// TIA Portal project "Pierwszy_Projekt_16022023" (V16)

(* hardware
DEVICE "S71500/ET200MP station_1"  S7-1500 station
   slot 0: "Rail_0"  Rack  6ES7 590-1***0-0AA0
   slot 1: "PLC_1"  CPU 1518F-4 PN/DP  6ES7 518-4FP00-3AB0  V2.8
      slot 3: "CPU display_1"  6ES7591-1BA00-0AA0
      slot 32768: "PROFINET interface_1"  X1
         slot 32769: "Port_1"  X1 P1
         slot 32770: "Port_2"  X1 P2
      slot 33024: "PROFINET interface_2"  X2
         slot 33025: "Port_1"  X2 P1
      slot 33280: "PROFINET interface GBIT_3"  X3
         slot 33281: "Port_1"  X3 P1
      slot 33536: "DP interface_1"  X4
      slot 34817: "Virtual CP interface port_1"  Virtual CP interface port  Virtual CP interface port
*)

// ===== PLC "PLC_1"  CPU 1518F-4 PN/DP =====

VAR_GLOBAL   // PLC tag table "Default tag table"
   "System_Byte" AT %MB1 : Byte;
   "FirstScan" AT %M1.0 : Bool;
   "DiagStatusUpdate" AT %M1.1 : Bool;
   "AlwaysTRUE" AT %M1.2 : Bool;
   "AlwaysFALSE" AT %M1.3 : Bool;
   "Clock_Byte" AT %MB0 : Byte;
   "Clock_10Hz" AT %M0.0 : Bool;
   "Clock_5Hz" AT %M0.1 : Bool;
   "Clock_2.5Hz" AT %M0.2 : Bool;
   "Clock_2Hz" AT %M0.3 : Bool;
   "Clock_1.25Hz" AT %M0.4 : Bool;
   "Clock_1Hz" AT %M0.5 : Bool;
   "Clock_0.625Hz" AT %M0.6 : Bool;
   "Clock_0.5Hz" AT %M0.7 : Bool;
   "11-PLC01-MANUAL" AT %Q1.6 : Bool;
   "11-PLC01-AUTOMAT" AT %Q1.7 : Bool;
   "11-PLC01-DISPLAY01" AT %QD58 : Real;
   "Tag_1" AT %QD40 : Real;
   "Tag_2" AT %Q2.5 : Bool;
   "Tag_3" AT %QD48 : Real;
   "Tag_4" AT %M2.0 : Bool;
   "Tag_5" AT %I4.4 : Bool;
   "Tag_6" AT %M3.0 : Bool;
   "Tag_7" AT %M3.1 : Bool;
   "Tag_8" AT %M3.2 : Bool;
END_VAR

VAR_GLOBAL   // PLC tag table "Tag table from XML_1"
   "11-PLC01-CNR01-SQ01" AT %I0.0 : Bool;
   "11-PLC01-CNR01-SQ02" AT %I0.1 : Bool;
   "11-PLC01-CNR01-ENC-A" AT %I0.2 : Bool;
   "11-PLC01-CNR01-ENC-B" AT %I0.3 : Bool;
   "11-PLC01-CNR02-SQ01" AT %I0.4 : Bool;
   "11-PLC01-CNR02-SQ02" AT %I0.5 : Bool;
   "11-PLC01-CNR02-ENC-A" AT %I0.6 : Bool;
   "11-PLC01-CNR02-ENC-B" AT %I0.7 : Bool;
   "11-PLC01-CNR03-SQ01" AT %I1.0 : Bool;
   "11-PLC01-CNR03-SQ02" AT %I1.1 : Bool;
   "11-PLC01-CNR03-ENC-A" AT %I1.2 : Bool;
   "11-PLC01-CNR03-ENC-B" AT %I1.3 : Bool;
   "11-PLC01-B01(START)" AT %I3.5 : Bool;
   "11-PLC01-B02(STOP)" AT %I3.6 : Bool;
   "11-PLC01-B03(RESET)" AT %I3.7 : Bool;
   "11-PLC01-B04(MANUAL)" AT %I4.0 : Bool;
   "11-PLC01-B05(AUTOMAT)" AT %I4.1 : Bool;
   "FACTORY I/O (Running)" AT %I4.2 : Bool;
   "FACTORY I/O (Paused)" AT %I4.3 : Bool;
   "FACTORY I/O (Reset)" AT %Q1.5 : Bool;
   "11-PLC01-PX01(START)" AT %Q0.0 : Bool;
   "11-PLC01-PX02(STOP)" AT %Q0.1 : Bool;
   "11-PLC01-PX03(RESET)" AT %Q0.2 : Bool;
   "11-PLC01-CNR01-EM01" AT %Q0.3 : Bool;
   "11-PLC01-CNR03-RE01" AT %Q0.4 : Bool;
   "FACTORY I/O (Run)" AT %Q1.3 : Bool;
   "FACTORY I/O (Pause)" AT %Q1.4 : Bool;
   "FACTORY I/O (Time Scale)" AT %ID34 : Real;
   "11-PLC01-CNR01" AT %QD30 : Real;
   "11-PLC01-CNR02" AT %QD34 : Real;
   "11-PLC01-CNR03" AT %QD38 : Real;
   "FACTORY I/O (Camera Position)" AT %QD54 : DInt;
   "11-PLC01-TT01-SQ01" AT %I1.4 : Bool;
   "11-PLC01-TT01-SQ02" AT %I1.5 : Bool;
   "11-PLC01-TT01-SQ03" AT %I1.6 : Bool;
   "11-PLC01-TT01-SQ04" AT %I1.7 : Bool;
   "11-PLC01-TT01-SQ05" AT %I2.0 : Bool;
   "11-PLC01-CNR04-SQ01" AT %I2.1 : Bool;
   "11-PLC01-CNR04-SQ02" AT %I2.2 : Bool;
   "11-PLC01-CNR04-ENC-A" AT %I2.3 : Bool;
   "11-PLC01-CNR04-ENC-B" AT %I2.4 : Bool;
   "11-PLC01-CNR05-SQ01" AT %I2.5 : Bool;
   "11-PLC01-CNR05-SQ02" AT %I2.6 : Bool;
   "11-PLC01-CNR05-ENC-A" AT %I2.7 : Bool;
   "11-PLC01-CNR05-ENC-B" AT %I3.0 : Bool;
   "11-PLC01-CNR06-SQ01" AT %I3.1 : Bool;
   "11-PLC01-CNR06-SQ02" AT %I3.2 : Bool;
   "11-PLC01-CNR06-ENC-A" AT %I3.3 : Bool;
   "11-PLC01-CNR06-ENC-B" AT %I3.4 : Bool;
   "11-PLC01-CNR04-RE01" AT %Q0.5 : Bool;
   "11-PLC01-CNR05-RE01" AT %Q0.6 : Bool;
   "11-PLC01-CNR06-RE01" AT %Q0.7 : Bool;
   "11-PLC01-TT01-LEFT" AT %Q2.0 : Bool;
   "11-PLC01-TT01-RIGHT" AT %Q2.1 : Bool;
   "11-PLC01-TT01-FORWARD" AT %Q2.2 : Bool;
   "11-PLC01-TT01-BACKWARD" AT %Q2.3 : Bool;
   "11-PLC01-CNR03-FLC01" AT %ID30 : Real;
   "11-PLC01-CNR04" AT %QD42 : Real;
   "11-PLC01-CNR05" AT %QD46 : Real;
   "11-PLC01-CNR06" AT %QD50 : Real;
END_VAR

DATA_BLOCK "Main_Safety_RTG1_DB"   // DB1, F_DB
{ S7_Optimized_Access := 'TRUE' }
NAME : FUSI
VERSION : 0.1
// stored: InstanceOfName Main_Safety_RTG1
"Main_Safety_RTG1"
BEGIN
END_DATA_BLOCK

DATA_BLOCK "IDB_11_CNR01"   // DB4
{ S7_Optimized_Access := 'TRUE' }
VERSION : 0.1
// stored: InstanceOfName FB_Conveyor
"FB_Conveyor"
BEGIN
END_DATA_BLOCK

DATA_BLOCK "IDB_11_CNR02"   // DB5
{ S7_Optimized_Access := 'TRUE' }
VERSION : 0.1
// stored: InstanceOfName FB_Conveyor
"FB_Conveyor"
BEGIN
END_DATA_BLOCK

DATA_BLOCK "DB_Manual"   // DB6
{ S7_Optimized_Access := 'TRUE' }
VERSION : 0.1
   VAR
      "11-CNR01-CONV" : Struct
         SelectManualMode : Bool := TRUE;
         StartStop : Bool := TRUE;
         SetSpeed : Int := 33;
      END_STRUCT;
      "11-CNR02-CONV" : Struct
         SelectManualMode : Bool := TRUE;
         StartStop : Bool := TRUE;
         SetSpeed : Int := 66;
      END_STRUCT;
      "11-CNR03-CONV" : Struct
         SelectManualMode : Bool := TRUE;
         StartStop : Bool := TRUE;
         SetSpeed : Int := 99;
      END_STRUCT;
   END_VAR
BEGIN
END_DATA_BLOCK

DATA_BLOCK "IDB_11_CNR03"   // DB7
{ S7_Optimized_Access := 'TRUE' }
VERSION : 0.1
// stored: InstanceOfName FB_Conveyor
"FB_Conveyor"
BEGIN
END_DATA_BLOCK

DATA_BLOCK "IDB_11_CNR01_VFD"   // DB8
{ S7_Optimized_Access := 'TRUE' }
VERSION : 0.1
// stored: InstanceOfName FB_Inverter
"FB_Inverter"
BEGIN
END_DATA_BLOCK

DATA_BLOCK "DB_Configuration"   // DB9
{ S7_Optimized_Access := 'TRUE' }
VERSION : 0.1
   VAR
      "11-CNR01-VFD_1" : Struct
         InterlockForward : Bool := TRUE;
         InterlockReverse : Bool := FALSE;
      END_STRUCT;
      "11-CNR02-VFD" : Struct
         InterlockForward : Bool := TRUE;
         InterlockReverse : Bool := FALSE;
      END_STRUCT;
      "11-CNR03-VFD" : Struct
         InterlockForward : Bool := TRUE;
         InterlockReverse : Bool := FALSE;
      END_STRUCT;
   END_VAR
BEGIN
END_DATA_BLOCK

DATA_BLOCK "DB_Signals"   // DB10
{ S7_Optimized_Access := 'TRUE' }
VERSION : 0.1
   VAR
      "11-CNR01-VFD" : Struct
         RunForward : Bool;
         RunReverse : Bool;
         ConveyorSpeedSetpoint : Real := 0.0;
      END_STRUCT;
      "11-CNR02-VFD" : Struct
         RunForward : Bool;
         RunReverse : Bool;
         ConveyorSpeedSetpoint : Real := 0.0;
      END_STRUCT;
      "11-CNR03-VFD" : Struct
         RunForward : Bool;
         RunReverse : Bool;
         ConveyorSpeedSetpoint : Real := 0.0;
      END_STRUCT;
   END_VAR
BEGIN
END_DATA_BLOCK

DATA_BLOCK "IDB_11_CNR02_VFD"   // DB11
{ S7_Optimized_Access := 'TRUE' }
VERSION : 0.1
// stored: InstanceOfName FB_Inverter
"FB_Inverter"
BEGIN
END_DATA_BLOCK

DATA_BLOCK "IDB_11_CNR03_VFD"   // DB12
{ S7_Optimized_Access := 'TRUE' }
VERSION : 0.1
// stored: InstanceOfName FB_Inverter
"FB_Inverter"
BEGIN
END_DATA_BLOCK

DATA_BLOCK "IDB_11_System"   // DB14
{ S7_Optimized_Access := 'TRUE' }
VERSION : 0.1
// stored: InstanceOfName FB_Control
"FB_Control"
BEGIN
END_DATA_BLOCK

DATA_BLOCK "DB_Control"   // DB15
{ S7_Optimized_Access := 'TRUE' }
VERSION : 0.1
   VAR
      StartCommand : Bool := TRUE;
      StopCommand : Bool;
      StartFeedback : Bool;
      StopFeedback : Bool;
      ManualFeedback : Bool;
   END_VAR
BEGIN
END_DATA_BLOCK

DATA_BLOCK "IDB_11_TurnTable"   // DB16
{ S7_Optimized_Access := 'TRUE' }
VERSION : 0.1
// stored: InstanceOfName FB_TurnTable
"FB_TurnTable"
BEGIN
END_DATA_BLOCK

DATA_BLOCK "DB_Chute"   // DB17
{ S7_Optimized_Access := 'TRUE' }
VERSION : 0.1
   VAR
      SmallPackage : Int;
      MediumPackage : Int;
      BigPackage : Int;
   END_VAR
BEGIN
END_DATA_BLOCK

DATA_BLOCK "IDB_Fifo"   // DB18
{ S7_Optimized_Access := 'TRUE' }
VERSION : 0.1
// stored: InstanceOfName FB_Fifo
"FB_Fifo"
BEGIN
END_DATA_BLOCK

DATA_BLOCK "DB_Fifo"   // DB19
{ S7_Optimized_Access := 'TRUE' }
VERSION : 0.1
   VAR
      Array_Destiny : Array[0..10] of Real;
      Array_Return : Int;
      Array_EndOfQueue : Array[0..10] of Real;
      Array_Input : Array[0..5] of Real;
   END_VAR
BEGIN
   Array_Destiny[0] := 0.0;
   Array_Destiny[1] := 0.0;
   Array_Destiny[2] := 0.0;
   Array_Destiny[3] := 0.0;
   Array_Destiny[4] := 0.0;
   Array_Destiny[5] := 0.0;
   Array_Destiny[6] := 0.0;
   Array_Destiny[7] := 0.0;
   Array_Destiny[8] := 0.0;
   Array_Destiny[9] := 0.0;
   Array_Destiny[10] := 0.0;
   Array_EndOfQueue[0] := 0.0;
   Array_EndOfQueue[1] := 0.0;
   Array_EndOfQueue[2] := 0.0;
   Array_EndOfQueue[3] := 0.0;
   Array_EndOfQueue[4] := 0.0;
   Array_EndOfQueue[5] := 0.0;
   Array_EndOfQueue[6] := 0.0;
   Array_EndOfQueue[7] := 0.0;
   Array_EndOfQueue[8] := 0.0;
   Array_EndOfQueue[9] := 0.0;
   Array_EndOfQueue[10] := 0.0;
   Array_Input[0] := 0.0;
   Array_Input[1] := 0.0;
   Array_Input[2] := 0.0;
   Array_Input[3] := 0.0;
   Array_Input[4] := 0.0;
   Array_Input[5] := 0.0;
END_DATA_BLOCK

DATA_BLOCK "IDB_11_CNRO4_AmountOfPackage"   // DB25
{ S7_Optimized_Access := 'TRUE' }
VERSION : 0.1
// stored: InstanceOfName FB_Chute
"FB_Chute"
BEGIN
END_DATA_BLOCK

// folder: System blocks/Program resources

DATA_BLOCK "StartButtonCount_DB"   // DB2
{ S7_Optimized_Access := 'TRUE' }
AUTHOR : Simatic
FAMILY : IEC
NAME : CNTR
VERSION : 1.0
// stored: InstanceOfName IEC_COUNTER
"IEC_COUNTER"
BEGIN
END_DATA_BLOCK

DATA_BLOCK "DelayStart_DB"   // DB3
{ S7_Optimized_Access := 'TRUE' }
AUTHOR : Simatic
FAMILY : IEC
NAME : IEC_TMR
VERSION : 1.0
// stored: InstanceOfName IEC_TIMER
"IEC_TIMER"
BEGIN
END_DATA_BLOCK

DATA_BLOCK "s_TON_Timer"   // DB13
{ S7_Optimized_Access := 'TRUE' }
AUTHOR : Simatic
FAMILY : IEC
NAME : IEC_TMR
VERSION : 1.0
// stored: InstanceOfName IEC_TIMER
"IEC_TIMER"
BEGIN
END_DATA_BLOCK

DATA_BLOCK "IDB_QueueCounter"   // DB21
{ S7_Optimized_Access := 'TRUE' }
AUTHOR : Simatic
FAMILY : IEC
NAME : CNTR
VERSION : 1.0
// stored: InstanceOfName IEC_COUNTER
"IEC_COUNTER"
BEGIN
END_DATA_BLOCK

DATA_BLOCK "IDB_QueueEndCounter"   // DB22
{ S7_Optimized_Access := 'TRUE' }
AUTHOR : Simatic
FAMILY : IEC
NAME : CNTR
VERSION : 1.0
// stored: InstanceOfName IEC_COUNTER
"IEC_COUNTER"
BEGIN
END_DATA_BLOCK

DATA_BLOCK "IEC_Counter_0_DB"   // DB23
{ S7_Optimized_Access := 'TRUE' }
AUTHOR : Simatic
FAMILY : IEC
NAME : CNTR
VERSION : 1.0
// stored: InstanceOfName IEC_COUNTER
"IEC_COUNTER"
BEGIN
END_DATA_BLOCK

DATA_BLOCK "IEC_Counter_0_DB_1"   // DB24
{ S7_Optimized_Access := 'TRUE' }
AUTHOR : Simatic
FAMILY : IEC
NAME : CNTR
VERSION : 1.0
// stored: InstanceOfName IEC_COUNTER
"IEC_COUNTER"
BEGIN
END_DATA_BLOCK

DATA_BLOCK "IEC_Counter_0_DB_2"   // DB26
{ S7_Optimized_Access := 'TRUE' }
AUTHOR : Simatic
FAMILY : IEC
NAME : CNTR
VERSION : 1.0
// stored: InstanceOfName IEC_COUNTER
"IEC_COUNTER"
BEGIN
END_DATA_BLOCK

// folder: (top level)

FUNCTION_BLOCK "Main_Safety_RTG1"   // FB1, F_FBD
{ S7_Optimized_Access := 'TRUE' }
BEGIN
END_FUNCTION_BLOCK

FUNCTION_BLOCK "FB_Conveyor"   // FB2, LAD
{ S7_Optimized_Access := 'TRUE' }
VERSION : 0.1
   VAR_INPUT
      ir_ConveyorSpeed : Real;
      ix_PEC_BOS : Bool;
      ix_PEC_EOS : Bool;
   END_VAR
   VAR_IN_OUT
      iqx_StartStop : Bool;
      iqi_SetSpeed : Int;
      iqx_SelectManualMode : Bool;
      iqx_InverterSpeedSetpoint : Real;
      iqx_InverterRunForward : Bool;
      iqx_InverterRunReverse : Bool;
      iqx_ControlStart : Bool;
      iqx_ControlStop : Bool;
      iqx_ControlManual : Bool;
      igx_ConvFlow : Bool;
   END_VAR
   VAR
      sx_Manual : Bool;
      sx_Automatic : Bool;
   END_VAR
   VAR_TEMP
      tr_SpeedProcent : Real;
   END_VAR
   VAR_TEMP   // added for the SCL form of the ladder/FBD networks
      _w1 : Bool;
      _w2 : Bool;
      _w3 : Bool;
   END_VAR
BEGIN

REGION Network 1: Manual mode
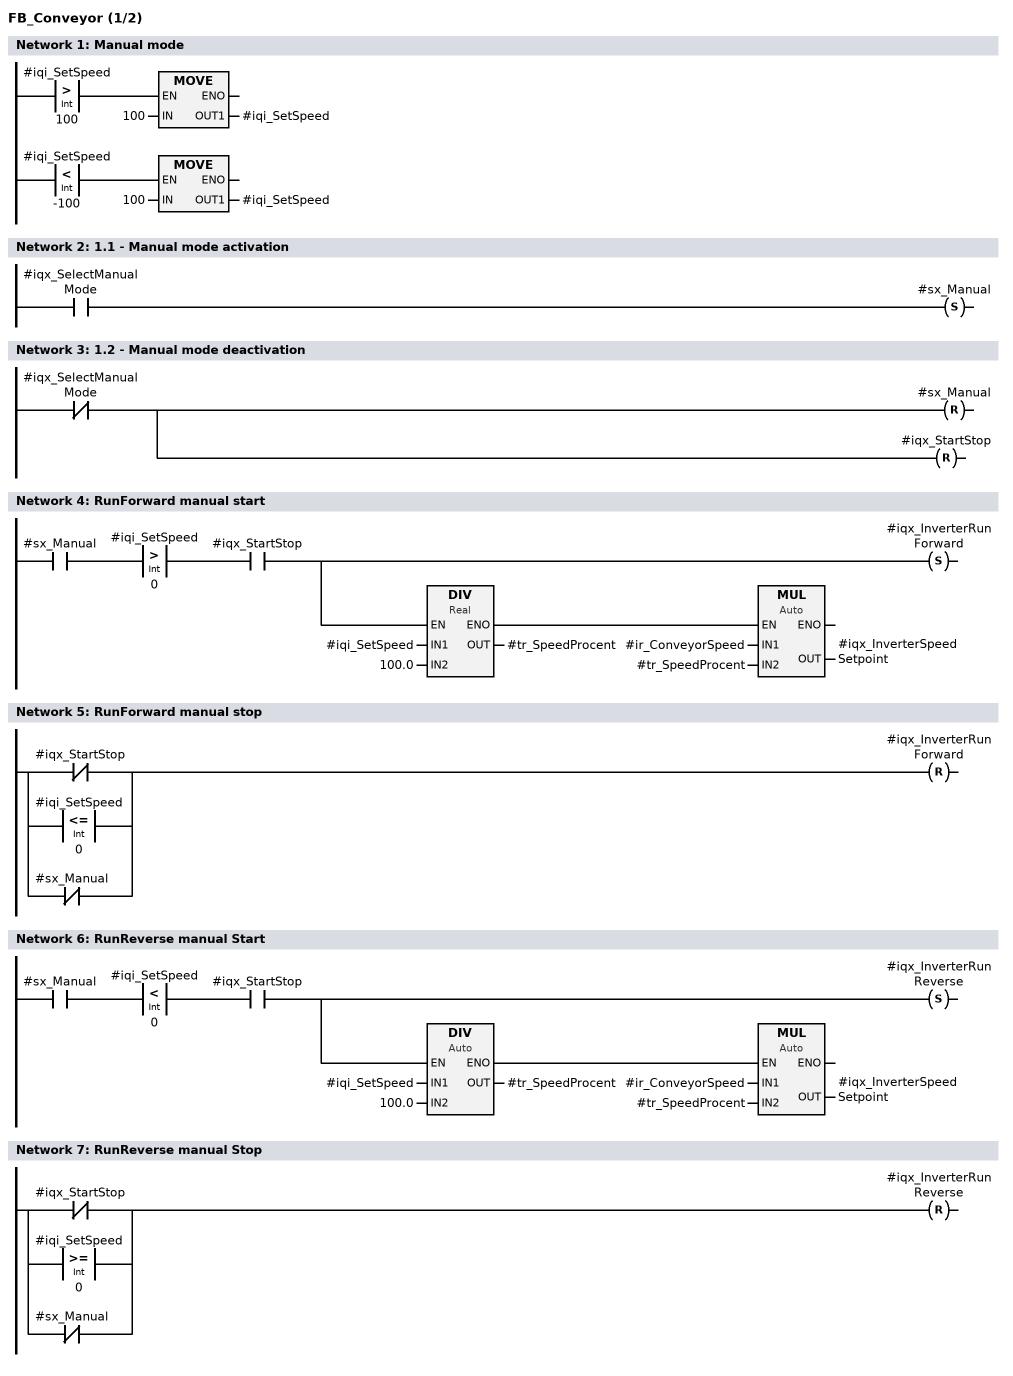
   RUNG wire#powerrail
      { S7_Templates := "SrcType := Int" } GT_Contact(in1 := #iqi_SetSpeed, in2 := 100)
      Move(in := 100, out1 => #iqi_SetSpeed)
   END_RUNG
   RUNG wire#powerrail
      { S7_Templates := "SrcType := Int" } LT_Contact(in1 := #iqi_SetSpeed, in2 := -100)
      Move(in := 100, out1 => #iqi_SetSpeed)
   END_RUNG
   // the same network as SCL:
   IF #iqi_SetSpeed > 100 THEN #iqi_SetSpeed := 100; END_IF;
   IF #iqi_SetSpeed < (-100) THEN #iqi_SetSpeed := 100; END_IF;
END_REGION

REGION Network 2: 1.1 - Manual mode activation
   RUNG wire#powerrail
      Contact( #iqx_SelectManualMode )
      S_Coil( #sx_Manual )
   END_RUNG
   // the same network as SCL:
   IF #iqx_SelectManualMode THEN #sx_Manual := TRUE; END_IF;
END_REGION

REGION Network 3: 1.2 - Manual mode deactivation
   RUNG wire#powerrail
      I_Contact( #iqx_SelectManualMode )
      wire#w1
      R_Coil( #sx_Manual )
   END_RUNG
   RUNG wire#w1
      R_Coil( #iqx_StartStop )
   END_RUNG
   // the same network as SCL:
   IF NOT #iqx_SelectManualMode THEN
       #sx_Manual := FALSE;
       #iqx_StartStop := FALSE;
   END_IF;
END_REGION

REGION Network 4: RunForward manual start
   RUNG wire#powerrail
      Contact( #sx_Manual )
      { S7_Templates := "SrcType := Int" } GT_Contact(in1 := #iqi_SetSpeed, in2 := 0)
      Contact( #iqx_StartStop )
      wire#w1
      S_Coil( #iqx_InverterRunForward )
   END_RUNG
   RUNG wire#w1
      { S7_Templates := "SrcType := Real" } Div(in1 := #iqi_SetSpeed, in2 := 100.0, out => #tr_SpeedProcent)
      Mul(in1 := #ir_ConveyorSpeed, in2 := #tr_SpeedProcent, out => #iqx_InverterSpeedSetpoint)
   END_RUNG
   // the same network as SCL:
   IF #sx_Manual AND (#iqi_SetSpeed > 0) AND #iqx_StartStop THEN
       #iqx_InverterRunForward := TRUE;
       #tr_SpeedProcent := #iqi_SetSpeed / 100.0;
       #iqx_InverterSpeedSetpoint := #ir_ConveyorSpeed * #tr_SpeedProcent;
   END_IF;
END_REGION

REGION Network 5: RunForward manual stop
   RUNG wire#powerrail
      I_Contact( #iqx_StartStop )
      wire#w1
      R_Coil( #iqx_InverterRunForward )
   END_RUNG
   RUNG wire#powerrail
      { S7_Templates := "SrcType := Int" } LE_Contact(in1 := #iqi_SetSpeed, in2 := 0)
   END_RUNG wire#w1
   RUNG wire#powerrail
      I_Contact( #sx_Manual )
   END_RUNG wire#w1
   // the same network as SCL:
   IF NOT #iqx_StartStop OR (#iqi_SetSpeed <= 0) OR NOT #sx_Manual THEN
       #iqx_InverterRunForward := FALSE;
   END_IF;
END_REGION

REGION Network 6: RunReverse manual Start
   RUNG wire#powerrail
      Contact( #sx_Manual )
      { S7_Templates := "SrcType := Int" } LT_Contact(in1 := #iqi_SetSpeed, in2 := 0)
      Contact( #iqx_StartStop )
      wire#w1
      S_Coil( #iqx_InverterRunReverse )
   END_RUNG
   RUNG wire#w1
      Div(in1 := #iqi_SetSpeed, in2 := 100.0, out => #tr_SpeedProcent)
      Mul(in1 := #ir_ConveyorSpeed, in2 := #tr_SpeedProcent, out => #iqx_InverterSpeedSetpoint)
   END_RUNG
   // the same network as SCL:
   IF #sx_Manual AND (#iqi_SetSpeed < 0) AND #iqx_StartStop THEN
       #iqx_InverterRunReverse := TRUE;
       #tr_SpeedProcent := #iqi_SetSpeed / 100.0;
       #iqx_InverterSpeedSetpoint := #ir_ConveyorSpeed * #tr_SpeedProcent;
   END_IF;
END_REGION

REGION Network 7: RunReverse manual Stop
   RUNG wire#powerrail
      I_Contact( #iqx_StartStop )
      wire#w1
      R_Coil( #iqx_InverterRunReverse )
   END_RUNG
   RUNG wire#powerrail
      { S7_Templates := "SrcType := Int" } GE_Contact(in1 := #iqi_SetSpeed, in2 := 0)
   END_RUNG wire#w1
   RUNG wire#powerrail
      I_Contact( #sx_Manual )
   END_RUNG wire#w1
   // the same network as SCL:
   IF NOT #iqx_StartStop OR (#iqi_SetSpeed >= 0) OR NOT #sx_Manual THEN
       #iqx_InverterRunReverse := FALSE;
   END_IF;
END_REGION

REGION Network 8: Automatic mode activation
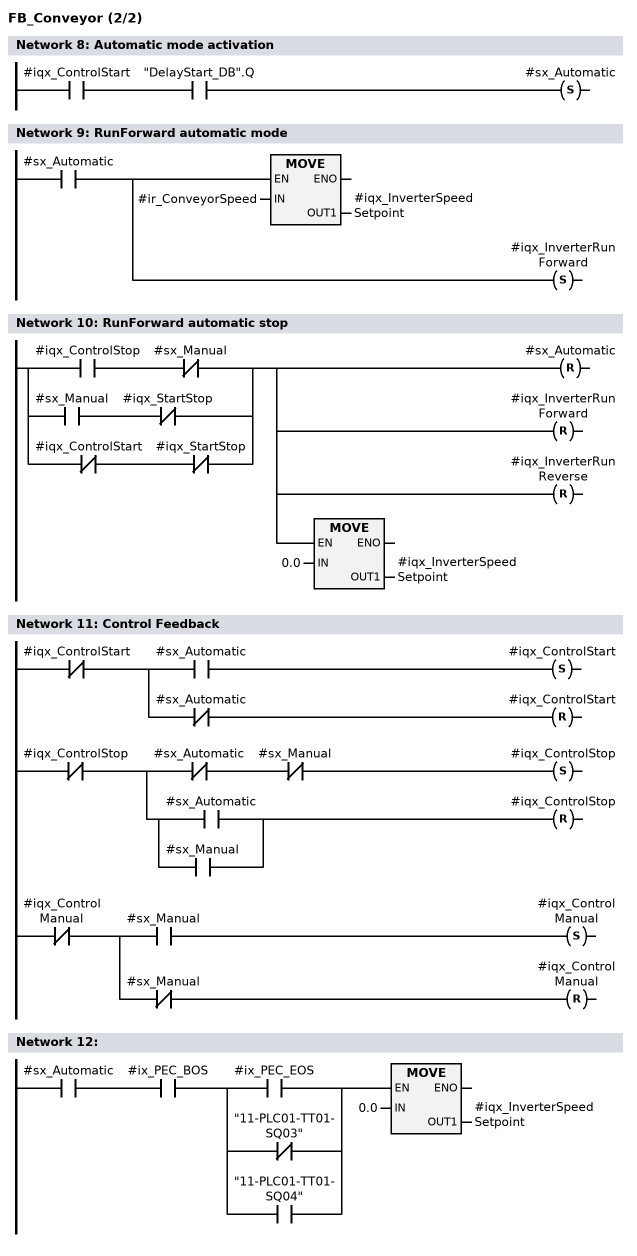
   RUNG wire#powerrail
      Contact( #iqx_ControlStart )
      Contact( "DelayStart_DB".Q )
      S_Coil( #sx_Automatic )
   END_RUNG
   // the same network as SCL:
   IF #iqx_ControlStart AND "DelayStart_DB".Q THEN #sx_Automatic := TRUE; END_IF;
END_REGION

REGION Network 9: RunForward automatic mode
   RUNG wire#powerrail
      Contact( #sx_Automatic )
      wire#w1
      Move(in := #ir_ConveyorSpeed, out1 => #iqx_InverterSpeedSetpoint)
   END_RUNG
   RUNG wire#w1
      S_Coil( #iqx_InverterRunForward )
   END_RUNG
   // the same network as SCL:
   IF #sx_Automatic THEN
       #iqx_InverterSpeedSetpoint := #ir_ConveyorSpeed;
       #iqx_InverterRunForward := TRUE;
   END_IF;
END_REGION

REGION Network 10: RunForward automatic stop
   RUNG wire#powerrail
      Contact( #iqx_ControlStop )
      I_Contact( #sx_Manual )
      wire#w1
      R_Coil( #sx_Automatic )
   END_RUNG
   RUNG wire#powerrail
      Contact( #sx_Manual )
      I_Contact( #iqx_StartStop )
   END_RUNG wire#w1
   RUNG wire#powerrail
      I_Contact( #iqx_ControlStart )
      I_Contact( #iqx_StartStop )
   END_RUNG wire#w1
   RUNG wire#w1
      R_Coil( #iqx_InverterRunForward )
   END_RUNG
   RUNG wire#w1
      R_Coil( #iqx_InverterRunReverse )
   END_RUNG
   RUNG wire#w1
      Move(in := 0.0, out1 => #iqx_InverterSpeedSetpoint)
   END_RUNG
   // the same network as SCL:
   IF (#iqx_ControlStop AND NOT #sx_Manual) OR (#sx_Manual AND NOT #iqx_StartStop) OR (NOT #iqx_ControlStart AND NOT #iqx_StartStop) THEN
       #sx_Automatic := FALSE;
       #iqx_InverterRunForward := FALSE;
       #iqx_InverterRunReverse := FALSE;
       #iqx_InverterSpeedSetpoint := 0.0;
   END_IF;
END_REGION

REGION Network 11: Control Feedback
   RUNG wire#powerrail
      I_Contact( #iqx_ControlStart )
      wire#w1
      Contact( #sx_Automatic )
      S_Coil( #iqx_ControlStart )
   END_RUNG
   RUNG wire#w1
      I_Contact( #sx_Automatic )
      R_Coil( #iqx_ControlStart )
   END_RUNG
   RUNG wire#powerrail
      I_Contact( #iqx_ControlStop )
      wire#w2
      I_Contact( #sx_Automatic )
      I_Contact( #sx_Manual )
      S_Coil( #iqx_ControlStop )
   END_RUNG
   RUNG wire#w2
      Contact( #sx_Automatic )
      wire#w3
      R_Coil( #iqx_ControlStop )
   END_RUNG
   RUNG wire#w2
      Contact( #sx_Manual )
   END_RUNG wire#w3
   RUNG wire#powerrail
      I_Contact( #iqx_ControlManual )
      wire#w4
      Contact( #sx_Manual )
      S_Coil( #iqx_ControlManual )
   END_RUNG
   RUNG wire#w4
      I_Contact( #sx_Manual )
      R_Coil( #iqx_ControlManual )
   END_RUNG
   // the same network as SCL:
   #_w1 := NOT #iqx_ControlStart;
   IF NOT #iqx_ControlStart AND #sx_Automatic THEN #iqx_ControlStart := TRUE; END_IF;
   IF #_w1 AND NOT #sx_Automatic THEN #iqx_ControlStart := FALSE; END_IF;
   #_w2 := NOT #iqx_ControlStop;
   IF NOT #iqx_ControlStop AND NOT #sx_Automatic AND NOT #sx_Manual THEN #iqx_ControlStop := TRUE; END_IF;
   IF #_w2 AND (#sx_Automatic OR #sx_Manual) THEN #iqx_ControlStop := FALSE; END_IF;
   #_w3 := NOT #iqx_ControlManual;
   IF NOT #iqx_ControlManual AND #sx_Manual THEN #iqx_ControlManual := TRUE; END_IF;
   IF #_w3 AND NOT #sx_Manual THEN #iqx_ControlManual := FALSE; END_IF;
END_REGION

REGION Network 12
   RUNG wire#powerrail
      Contact( #sx_Automatic )
      Contact( #ix_PEC_BOS )
      wire#w1
      Contact( #ix_PEC_EOS )
      wire#w2
      Move(in := 0.0, out1 => #iqx_InverterSpeedSetpoint)
   END_RUNG
   RUNG wire#w1
      I_Contact( "11-PLC01-TT01-SQ03" )
   END_RUNG wire#w2
   RUNG wire#w1
      Contact( "11-PLC01-TT01-SQ04" )
   END_RUNG wire#w2
   // the same network as SCL:
   IF #sx_Automatic AND #ix_PEC_BOS AND (#ix_PEC_EOS OR NOT "11-PLC01-TT01-SQ03" OR "11-PLC01-TT01-SQ04") THEN
       #iqx_InverterSpeedSetpoint := 0.0;
   END_IF;
END_REGION
END_FUNCTION_BLOCK

FUNCTION_BLOCK "FB_Inverter"   // FB3, LAD
{ S7_Optimized_Access := 'TRUE' }
VERSION : 0.1
   VAR_INPUT
      ix_InterlockForward : Bool;
      Ix_InterlockReverse : Bool;
      Ir_ConveyorSpeedSetpoint : Real;
   END_VAR
   VAR_OUTPUT
      qr_InverterSpeed : Real;
   END_VAR
   VAR_IN_OUT
      iqx_InverterRunForward : Bool;
      iqx_InverterRunReverse : Bool;
   END_VAR
   VAR
      sx_RunForward : Bool;
      sx_RunReverse : Bool;
   END_VAR
BEGIN

REGION Network 1: RunForward command
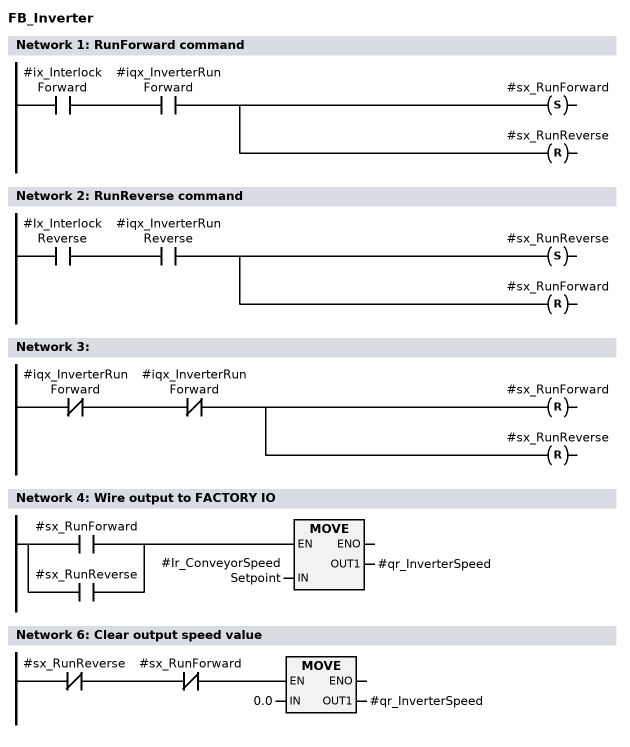
   RUNG wire#powerrail
      Contact( #ix_InterlockForward )
      Contact( #iqx_InverterRunForward )
      wire#w1
      S_Coil( #sx_RunForward )
   END_RUNG
   RUNG wire#w1
      R_Coil( #sx_RunReverse )
   END_RUNG
   // the same network as SCL:
   IF #ix_InterlockForward AND #iqx_InverterRunForward THEN
       #sx_RunForward := TRUE;
       #sx_RunReverse := FALSE;
   END_IF;
END_REGION

REGION Network 2: RunReverse command
   RUNG wire#powerrail
      Contact( #Ix_InterlockReverse )
      Contact( #iqx_InverterRunReverse )
      wire#w1
      S_Coil( #sx_RunReverse )
   END_RUNG
   RUNG wire#w1
      R_Coil( #sx_RunForward )
   END_RUNG
   // the same network as SCL:
   IF #Ix_InterlockReverse AND #iqx_InverterRunReverse THEN
       #sx_RunReverse := TRUE;
       #sx_RunForward := FALSE;
   END_IF;
END_REGION

REGION Network 3
   RUNG wire#powerrail
      I_Contact( #iqx_InverterRunForward )
      I_Contact( #iqx_InverterRunForward )
      wire#w1
      R_Coil( #sx_RunForward )
   END_RUNG
   RUNG wire#w1
      R_Coil( #sx_RunReverse )
   END_RUNG
   // the same network as SCL:
   IF NOT #iqx_InverterRunForward AND NOT #iqx_InverterRunForward THEN
       #sx_RunForward := FALSE;
       #sx_RunReverse := FALSE;
   END_IF;
END_REGION

REGION Network 4: Wire output to FACTORY IO
   RUNG wire#powerrail
      Contact( #sx_RunForward )
      wire#w1
      Move(in := #Ir_ConveyorSpeedSetpoint, out1 => #qr_InverterSpeed)
   END_RUNG
   RUNG wire#powerrail
      Contact( #sx_RunReverse )
   END_RUNG wire#w1
   // the same network as SCL:
   IF #sx_RunForward OR #sx_RunReverse THEN #qr_InverterSpeed := #Ir_ConveyorSpeedSetpoint; END_IF;
END_REGION

REGION Network 6: Clear output speed value
   RUNG wire#powerrail
      I_Contact( #sx_RunReverse )
      I_Contact( #sx_RunForward )
      Move(in := 0.0, out1 => #qr_InverterSpeed)
   END_RUNG
   // the same network as SCL:
   IF NOT #sx_RunReverse AND NOT #sx_RunForward THEN #qr_InverterSpeed := 0.0; END_IF;
END_REGION
END_FUNCTION_BLOCK

FUNCTION_BLOCK "FB_Control"   // FB4, LAD
{ S7_Optimized_Access := 'TRUE' }
VERSION : 0.1
   VAR_IN_OUT
      iqx_StartHMICommand : Bool;
      iqx_StartFeedback : Bool;
      iqx_ManualFeedback : Bool;
      iqx_StopHMICommand : Bool;
      iqx_StopFeedback : Bool;
   END_VAR
   VAR
      sudi_SignalingTime : Time := T#3000MS;
      sx_StartRequest : Bool;
      s_TON_Timer : TON_TIME;
   END_VAR
BEGIN

REGION Network 1: Start Request
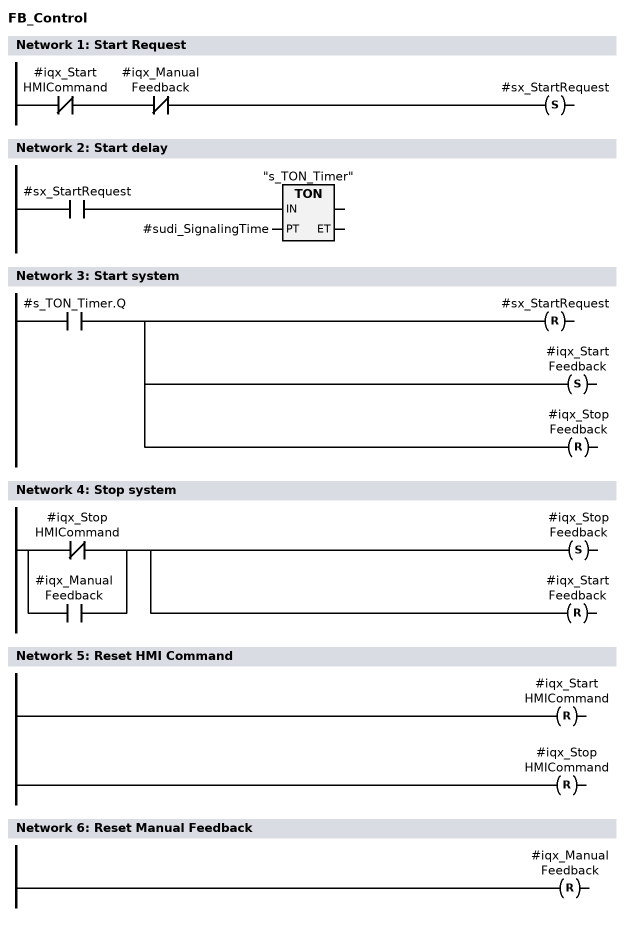
   RUNG wire#powerrail
      I_Contact( #iqx_StartHMICommand )
      I_Contact( #iqx_ManualFeedback )
      S_Coil( #sx_StartRequest )
   END_RUNG
   // the same network as SCL:
   IF NOT #iqx_StartHMICommand AND NOT #iqx_ManualFeedback THEN #sx_StartRequest := TRUE; END_IF;
END_REGION

REGION Network 2: Start delay
   "s_TON_Timer".TON(IN := #sx_StartRequest, PT := #sudi_SignalingTime);
END_REGION

REGION Network 3: Start system
   RUNG wire#powerrail
      Contact( #s_TON_Timer.Q )
      wire#w1
      R_Coil( #sx_StartRequest )
   END_RUNG
   RUNG wire#w1
      S_Coil( #iqx_StartFeedback )
   END_RUNG
   RUNG wire#w1
      R_Coil( #iqx_StopFeedback )
   END_RUNG
   // the same network as SCL:
   IF #s_TON_Timer.Q THEN
       #sx_StartRequest := FALSE;
       #iqx_StartFeedback := TRUE;
       #iqx_StopFeedback := FALSE;
   END_IF;
END_REGION

REGION Network 4: Stop system
   RUNG wire#powerrail
      I_Contact( #iqx_StopHMICommand )
      wire#w1
      S_Coil( #iqx_StopFeedback )
   END_RUNG
   RUNG wire#powerrail
      Contact( #iqx_ManualFeedback )
   END_RUNG wire#w1
   RUNG wire#w1
      R_Coil( #iqx_StartFeedback )
   END_RUNG
   // the same network as SCL:
   IF NOT #iqx_StopHMICommand OR #iqx_ManualFeedback THEN
       #iqx_StopFeedback := TRUE;
       #iqx_StartFeedback := FALSE;
   END_IF;
END_REGION

REGION Network 5: Reset HMI Command
   RUNG wire#powerrail
      R_Coil( #iqx_StartHMICommand )
   END_RUNG
   RUNG wire#powerrail
      R_Coil( #iqx_StopHMICommand )
   END_RUNG
   // the same network as SCL:
   #iqx_StartHMICommand := FALSE;
   #iqx_StopHMICommand := FALSE;
END_REGION

REGION Network 6: Reset Manual Feedback
   RUNG wire#powerrail
      R_Coil( #iqx_ManualFeedback )
   END_RUNG
   // the same network as SCL:
   #iqx_ManualFeedback := FALSE;
END_REGION
END_FUNCTION_BLOCK

FUNCTION_BLOCK "FB_TurnTable"   // FB5, LAD
{ S7_Optimized_Access := 'TRUE' }
VERSION : 0.1
   VAR_INPUT
      ix_turnTableSQ1 : Bool;
      ix_turnTableSQ2 : Bool;
      ix_0degree : Bool;
      ix_90degree : Bool;
      ix_packageDetect : Bool;
      ix_packageSmallPackageDetect : Bool;
      ix_packageMediumDetect : Bool;
      ix_packageBigDetect : Bool;
   END_VAR
   VAR_OUTPUT
      qx_Forward : Bool;
      qx_Backward : Bool;
      qx_Left : Bool;
      qx_Right : Bool;
      qx_CNR04 : Real;
      qx_CNR05 : Real;
      qx_CNR06 : Real;
   END_VAR
   VAR_IN_OUT
      iqx_automatic : Bool;
      iqx_Size : Real;
   END_VAR
   VAR
      sx_medium : Bool;
      sx_small : Bool;
      sx_Big : Bool;
      sx_left : Bool;
      sx_right : Bool;
      sx_leftB : Bool;
      sx_rightB : Bool;
      sx_rightC : Bool;
      sx_leftC : Bool;
   END_VAR
   VAR_TEMP   // added for the SCL form of the ladder/FBD networks
      _w1 : Bool;
   END_VAR
BEGIN

REGION Network 1: ActivationAutomaticMode
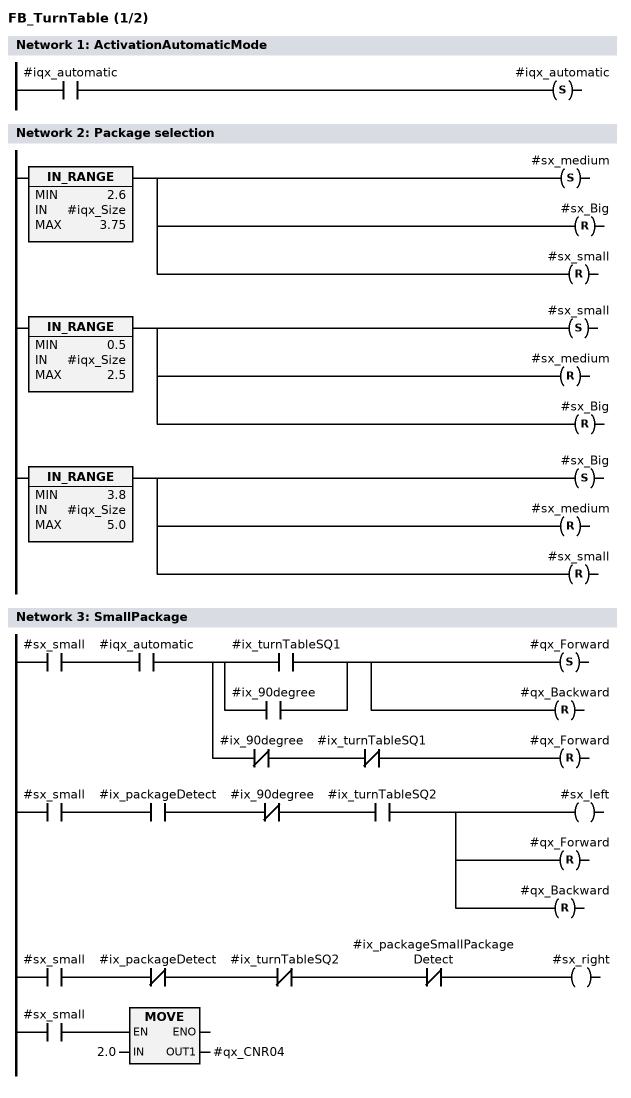
   RUNG wire#powerrail
      Contact( #iqx_automatic )
      S_Coil( #iqx_automatic )
   END_RUNG
   // the same network as SCL:
   IF #iqx_automatic THEN #iqx_automatic := TRUE; END_IF;
END_REGION

REGION Network 2: Package selection
   RUNG wire#powerrail
      { S7_Templates := "SrcType := Real" } InRange(min := 2.6, in := #iqx_Size, max := 3.75)
      wire#w1
      S_Coil( #sx_medium )
   END_RUNG
   RUNG wire#w1
      R_Coil( #sx_Big )
   END_RUNG
   RUNG wire#w1
      R_Coil( #sx_small )
   END_RUNG
   RUNG wire#powerrail
      { S7_Templates := "SrcType := Real" } InRange(min := 0.5, in := #iqx_Size, max := 2.5)
      wire#w2
      S_Coil( #sx_small )
   END_RUNG
   RUNG wire#w2
      R_Coil( #sx_medium )
   END_RUNG
   RUNG wire#w2
      R_Coil( #sx_Big )
   END_RUNG
   RUNG wire#powerrail
      { S7_Templates := "SrcType := Real" } InRange(min := 3.8, in := #iqx_Size, max := 5.0)
      wire#w3
      S_Coil( #sx_Big )
   END_RUNG
   RUNG wire#w3
      R_Coil( #sx_medium )
   END_RUNG
   RUNG wire#w3
      R_Coil( #sx_small )
   END_RUNG
   // the same network as SCL:
   IF (2.6 <= #iqx_Size) AND (#iqx_Size <= 3.75) THEN
       #sx_medium := TRUE;
       #sx_Big := FALSE;
       #sx_small := FALSE;
   END_IF;
   IF (0.5 <= #iqx_Size) AND (#iqx_Size <= 2.5) THEN
       #sx_small := TRUE;
       #sx_medium := FALSE;
       #sx_Big := FALSE;
   END_IF;
   IF (3.8 <= #iqx_Size) AND (#iqx_Size <= 5.0) THEN
       #sx_Big := TRUE;
       #sx_medium := FALSE;
       #sx_small := FALSE;
   END_IF;
END_REGION

REGION Network 3: SmallPackage
   RUNG wire#powerrail
      Contact( #sx_small )
      Contact( #iqx_automatic )
      wire#w1
      Contact( #ix_turnTableSQ1 )
      wire#w2
      S_Coil( #qx_Forward )
   END_RUNG
   RUNG wire#w1
      Contact( #ix_90degree )
   END_RUNG wire#w2
   RUNG wire#w2
      R_Coil( #qx_Backward )
   END_RUNG
   RUNG wire#w1
      I_Contact( #ix_90degree )
      I_Contact( #ix_turnTableSQ1 )
      R_Coil( #qx_Forward )
   END_RUNG
   RUNG wire#powerrail
      Contact( #sx_small )
      Contact( #ix_packageDetect )
      I_Contact( #ix_90degree )
      Contact( #ix_turnTableSQ2 )
      wire#w3
      Coil( #sx_left )
   END_RUNG
   RUNG wire#w3
      R_Coil( #qx_Forward )
   END_RUNG
   RUNG wire#w3
      R_Coil( #qx_Backward )
   END_RUNG
   RUNG wire#powerrail
      Contact( #sx_small )
      I_Contact( #ix_packageDetect )
      I_Contact( #ix_turnTableSQ2 )
      I_Contact( #ix_packageSmallPackageDetect )
      Coil( #sx_right )
   END_RUNG
   RUNG wire#powerrail
      Contact( #sx_small )
      Move(in := 2.0, out1 => #qx_CNR04)
   END_RUNG
   // the same network as SCL:
   #_w1 := #sx_small AND #iqx_automatic;
   IF #_w1 AND (#ix_turnTableSQ1 OR #ix_90degree) THEN
       #qx_Forward := TRUE;
       #qx_Backward := FALSE;
   END_IF;
   IF #_w1 AND NOT #ix_90degree AND NOT #ix_turnTableSQ1 THEN #qx_Forward := FALSE; END_IF;
   #sx_left := #sx_small AND #ix_packageDetect AND NOT #ix_90degree AND #ix_turnTableSQ2;
   IF #sx_left THEN
       #qx_Forward := FALSE;
       #qx_Backward := FALSE;
   END_IF;
   #sx_right := #sx_small AND NOT #ix_packageDetect AND NOT #ix_turnTableSQ2 AND NOT #ix_packageSmallPackageDetect;
   IF #sx_small THEN #qx_CNR04 := 2.0; END_IF;
END_REGION

REGION Network 4: MediumPackage
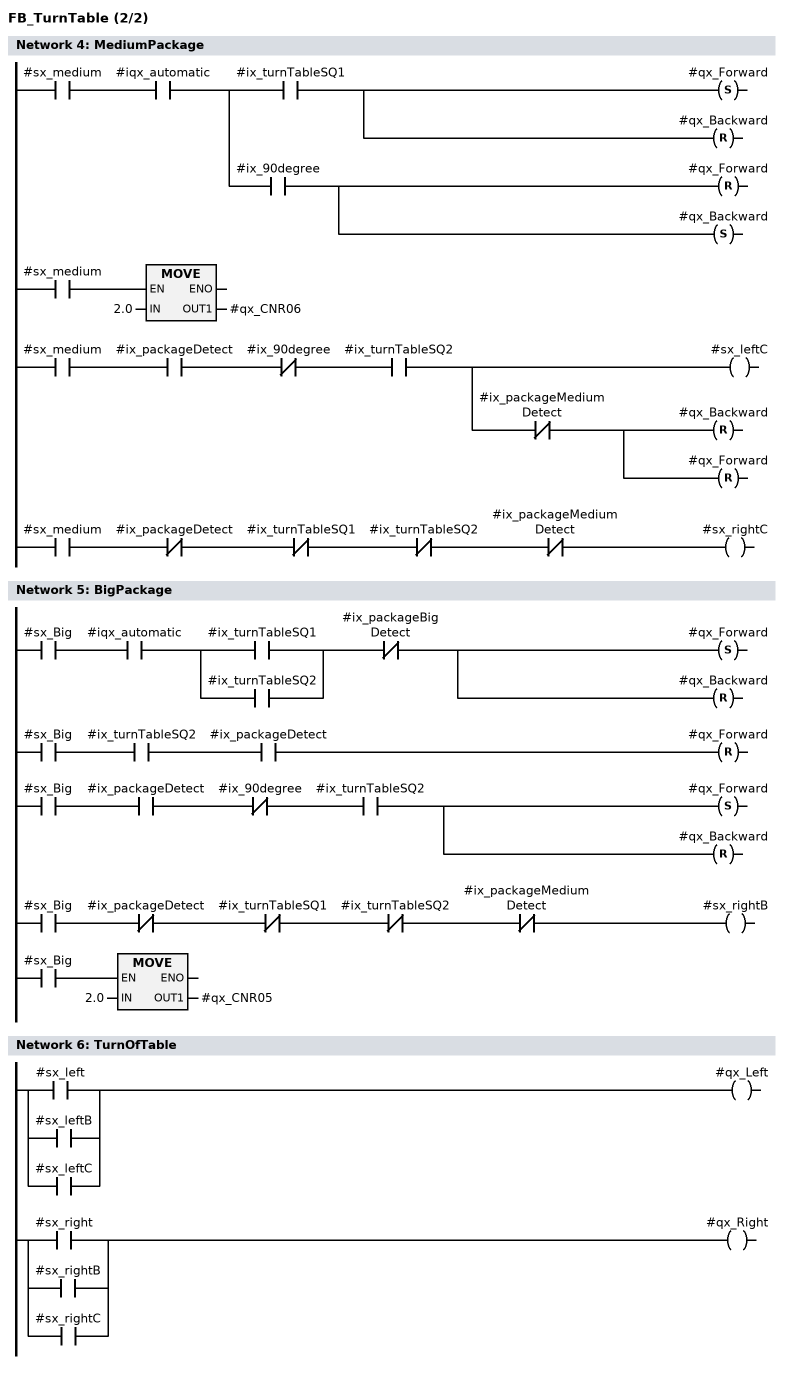
   RUNG wire#powerrail
      Contact( #sx_medium )
      Contact( #iqx_automatic )
      wire#w1
      Contact( #ix_turnTableSQ1 )
      wire#w2
      S_Coil( #qx_Forward )
   END_RUNG
   RUNG wire#w2
      R_Coil( #qx_Backward )
   END_RUNG
   RUNG wire#w1
      Contact( #ix_90degree )
      wire#w3
      R_Coil( #qx_Forward )
   END_RUNG
   RUNG wire#w3
      S_Coil( #qx_Backward )
   END_RUNG
   RUNG wire#powerrail
      Contact( #sx_medium )
      Move(in := 2.0, out1 => #qx_CNR06)
   END_RUNG
   RUNG wire#powerrail
      Contact( #sx_medium )
      Contact( #ix_packageDetect )
      I_Contact( #ix_90degree )
      Contact( #ix_turnTableSQ2 )
      wire#w4
      Coil( #sx_leftC )
   END_RUNG
   RUNG wire#w4
      I_Contact( #ix_packageMediumDetect )
      wire#w5
      R_Coil( #qx_Backward )
   END_RUNG
   RUNG wire#w5
      R_Coil( #qx_Forward )
   END_RUNG
   RUNG wire#powerrail
      Contact( #sx_medium )
      I_Contact( #ix_packageDetect )
      I_Contact( #ix_turnTableSQ1 )
      I_Contact( #ix_turnTableSQ2 )
      I_Contact( #ix_packageMediumDetect )
      Coil( #sx_rightC )
   END_RUNG
   // the same network as SCL:
   #_w1 := #sx_medium AND #iqx_automatic;
   IF #_w1 AND #ix_turnTableSQ1 THEN
       #qx_Forward := TRUE;
       #qx_Backward := FALSE;
   END_IF;
   IF #_w1 AND #ix_90degree THEN
       #qx_Forward := FALSE;
       #qx_Backward := TRUE;
   END_IF;
   IF #sx_medium THEN #qx_CNR06 := 2.0; END_IF;
   #sx_leftC := #sx_medium AND #ix_packageDetect AND NOT #ix_90degree AND #ix_turnTableSQ2;
   IF #sx_leftC AND NOT #ix_packageMediumDetect THEN
       #qx_Backward := FALSE;
       #qx_Forward := FALSE;
   END_IF;
   #sx_rightC := #sx_medium AND NOT #ix_packageDetect AND NOT #ix_turnTableSQ1 AND NOT #ix_turnTableSQ2 AND NOT #ix_packageMediumDetect;
END_REGION

REGION Network 5: BigPackage
   RUNG wire#powerrail
      Contact( #sx_Big )
      Contact( #iqx_automatic )
      wire#w1
      Contact( #ix_turnTableSQ1 )
      wire#w2
      I_Contact( #ix_packageBigDetect )
      wire#w3
      S_Coil( #qx_Forward )
   END_RUNG
   RUNG wire#w1
      Contact( #ix_turnTableSQ2 )
   END_RUNG wire#w2
   RUNG wire#w3
      R_Coil( #qx_Backward )
   END_RUNG
   RUNG wire#powerrail
      Contact( #sx_Big )
      Contact( #ix_turnTableSQ2 )
      Contact( #ix_packageDetect )
      R_Coil( #qx_Forward )
   END_RUNG
   RUNG wire#powerrail
      Contact( #sx_Big )
      Contact( #ix_packageDetect )
      I_Contact( #ix_90degree )
      Contact( #ix_turnTableSQ2 )
      wire#w4
      S_Coil( #qx_Forward )
   END_RUNG
   RUNG wire#w4
      R_Coil( #qx_Backward )
   END_RUNG
   RUNG wire#powerrail
      Contact( #sx_Big )
      I_Contact( #ix_packageDetect )
      I_Contact( #ix_turnTableSQ1 )
      I_Contact( #ix_turnTableSQ2 )
      I_Contact( #ix_packageMediumDetect )
      Coil( #sx_rightB )
   END_RUNG
   RUNG wire#powerrail
      Contact( #sx_Big )
      Move(in := 2.0, out1 => #qx_CNR05)
   END_RUNG
   // the same network as SCL:
   IF #sx_Big AND #iqx_automatic AND (#ix_turnTableSQ1 OR #ix_turnTableSQ2) AND NOT #ix_packageBigDetect THEN
       #qx_Forward := TRUE;
       #qx_Backward := FALSE;
   END_IF;
   IF #sx_Big AND #ix_turnTableSQ2 AND #ix_packageDetect THEN #qx_Forward := FALSE; END_IF;
   IF #sx_Big AND #ix_packageDetect AND NOT #ix_90degree AND #ix_turnTableSQ2 THEN
       #qx_Forward := TRUE;
       #qx_Backward := FALSE;
   END_IF;
   #sx_rightB := #sx_Big AND NOT #ix_packageDetect AND NOT #ix_turnTableSQ1 AND NOT #ix_turnTableSQ2 AND NOT #ix_packageMediumDetect;
   IF #sx_Big THEN #qx_CNR05 := 2.0; END_IF;
END_REGION

REGION Network 6: TurnOfTable
   RUNG wire#powerrail
      Contact( #sx_left )
      wire#w1
      Coil( #qx_Left )
   END_RUNG
   RUNG wire#powerrail
      Contact( #sx_leftB )
   END_RUNG wire#w1
   RUNG wire#powerrail
      Contact( #sx_leftC )
   END_RUNG wire#w1
   RUNG wire#powerrail
      Contact( #sx_right )
      wire#w2
      Coil( #qx_Right )
   END_RUNG
   RUNG wire#powerrail
      Contact( #sx_rightB )
   END_RUNG wire#w2
   RUNG wire#powerrail
      Contact( #sx_rightC )
   END_RUNG wire#w2
   // the same network as SCL:
   #qx_Left := #sx_left OR #sx_leftB OR #sx_leftC;
   #qx_Right := #sx_right OR #sx_rightB OR #sx_rightC;
END_REGION

REGION Network 7: StoppingUnusedConveyor
END_REGION
END_FUNCTION_BLOCK

FUNCTION_BLOCK "FB_Fifo"   // FB6, LAD
{ S7_Optimized_Access := 'TRUE' }
VERSION : 0.1
   VAR_OUTPUT
      Output_2 : Real;
   END_VAR
   VAR
      sx_Measure : Bool;
   END_VAR
   VAR_TEMP   // added for the SCL form of the ladder/FBD networks
      _w1 : Bool;
   END_VAR
BEGIN

REGION Network 1
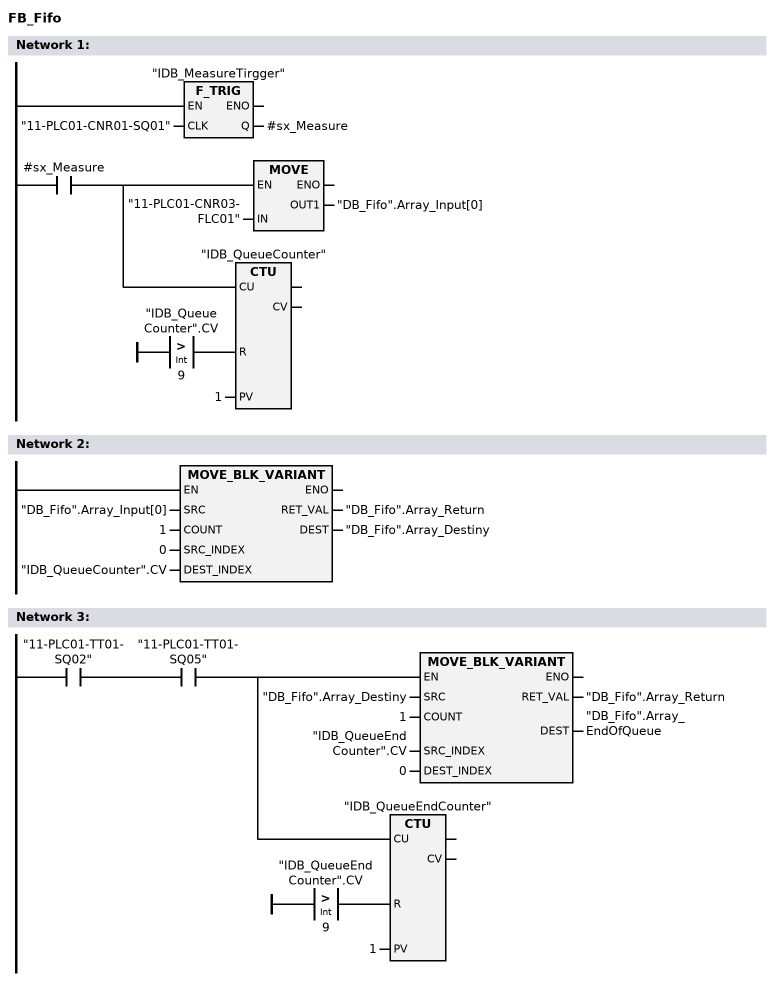
   "IDB_MeasureTirgger"(CLK := "11-PLC01-CNR01-SQ01", Q => #sx_Measure);   // F_TRIG
   IF #sx_Measure THEN "DB_Fifo".Array_Input[0] := "11-PLC01-CNR03-FLC01"; END_IF;
   "IDB_QueueCounter".CTU(CU := #sx_Measure, R := "IDB_QueueCounter".CV > 9, PV := 1);
END_REGION

REGION Network 2
   "DB_Fifo".Array_Return := MOVE_BLK_VARIANT(SRC := "DB_Fifo".Array_Input[0],
                           COUNT := 1,
                           SRC_INDEX := 0,
                           DEST_INDEX := "IDB_QueueCounter".CV,
                           DEST => "DB_Fifo".Array_Destiny);
END_REGION

REGION Network 3
   #_w1 := "11-PLC01-TT01-SQ02" AND "11-PLC01-TT01-SQ05";
   IF #_w1 THEN
       "DB_Fifo".Array_Return := MOVE_BLK_VARIANT(SRC := "DB_Fifo".Array_Destiny,
                               COUNT := 1,
                               SRC_INDEX := "IDB_QueueEndCounter".CV,
                               DEST_INDEX := 0,
                               DEST => "DB_Fifo".Array_EndOfQueue);
   END_IF;
   "IDB_QueueEndCounter".CTU(CU := #_w1, R := "IDB_QueueEndCounter".CV > 9, PV := 1);
END_REGION
END_FUNCTION_BLOCK

FUNCTION_BLOCK "FB_Chute"   // FB7, LAD
{ S7_Optimized_Access := 'TRUE' }
VERSION : 0.1
   VAR_INPUT
      ix_reset : Bool;
      ix_packageDetectSmall_1 : Bool;
      ix_packageDetectMedium_1 : Bool;
      ix_packageDetectBig_1 : Bool;
   END_VAR
   VAR_OUTPUT
      qi_amountSP : Int;
      qi_amountMP : Int;
      qi_amountBP : Int;
   END_VAR
BEGIN

REGION Network 2: small
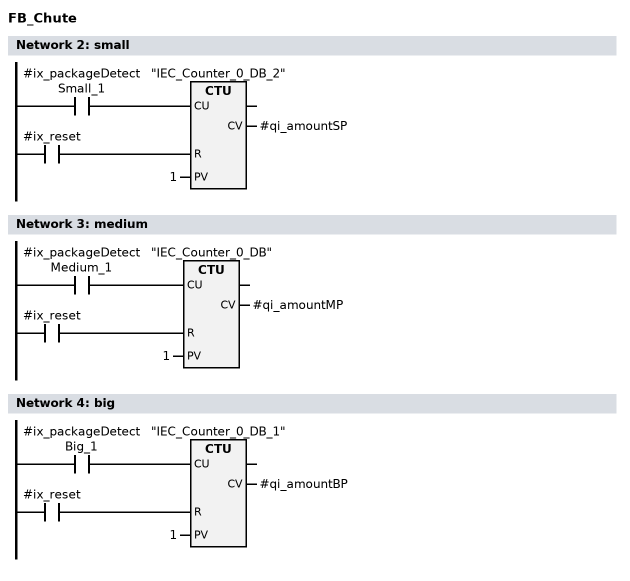
   "IEC_Counter_0_DB_2".CTU(CU := #ix_packageDetectSmall_1, R := #ix_reset, PV := 1, CV => #qi_amountSP);
END_REGION

REGION Network 3: medium
   "IEC_Counter_0_DB".CTU(CU := #ix_packageDetectMedium_1, R := #ix_reset, PV := 1, CV => #qi_amountMP);
END_REGION

REGION Network 4: big
   "IEC_Counter_0_DB_1".CTU(CU := #ix_packageDetectBig_1, R := #ix_reset, PV := 1, CV => #qi_amountBP);
END_REGION
END_FUNCTION_BLOCK

FUNCTION_BLOCK "FB_Sequence"   // FB8, GRAPH_PLUS
{ S7_Optimized_Access := 'TRUE' }
VERSION : 0.1
   VAR_INPUT
      OFF_SQ : Bool := false;   // Turn sequence off
      INIT_SQ : Bool := false;   // Set sequence to initial state
      ACK_EF : Bool := false;   // Acknowledge all errors and faults
      S_PREV : Bool := false;   // Output previous step in parameter S_NO
      S_NEXT : Bool := false;   // Indicate next step in parameter S_NO
      SW_AUTO : Bool := false;   // Automatic mode
      SW_TAP : Bool := false;   // Semiautomatic/switch with transition
      SW_TOP : Bool := false;   // Semiautomatic/ignore transition
      SW_MAN : Bool := false;   // Manual mode
      S_SEL : Int := 0;   // Select step to be output to S_NO
      S_ON : Bool := false;   // Activate step indicated in S_NO
      S_OFF : Bool := false;   // Deactivate step indicated S_NO
      T_PUSH : Bool := false;   // Enable transition to switch in semi automatic mode
   END_VAR
   VAR_OUTPUT
      S_NO : Int := 0;   // Step number
      S_MORE : Bool := false;   // More steps are available and can be shown in S_NO
      S_ACTIVE : Bool := false;   // Step indicated in S_NO is active
      ERR_FLT : Bool := false;   // Interlock or supervision group error
      AUTO_ON : Bool := false;   // Automatic mode is active
      TAP_ON : Bool := false;   // Semiautomatic mode/step with transition enabled
      TOP_ON : Bool := false;   // Semiautomatic mode/ignore transition enabled
      MAN_ON : Bool := false;   // Manual mode is active
   END_VAR
   VAR
      HMI_INFO : Array[0..0] of UInt;
      RT_DATA : G7_RTDataPlus_V6;   // Internal data area
      Trans1 : G7_TransitionPlus_V6;   // Transition structure
      Step1 : G7_StepPlus_V6;   // Step structure
      Step2 : G7_StepPlus_V6;   // Step structure
      Trans2 : G7_TransitionPlus_V6;   // Transition structure
      Step3 : G7_StepPlus_V6;   // Step structure
      Trans3 : G7_TransitionPlus_V6;   // Transition structure
      Step4 : G7_StepPlus_V6;   // Step structure
      Trans4 : G7_TransitionPlus_V6;   // Transition structure
      Step5 : G7_StepPlus_V6;   // Step structure
      Trans5 : G7_TransitionPlus_V6;   // Transition structure
      Step6 : G7_StepPlus_V6;   // Step structure
      Trans6 : G7_TransitionPlus_V6;   // Transition structure
      Step7 : G7_StepPlus_V6;   // Step structure
      Trans7 : G7_TransitionPlus_V6;   // Transition structure
      Step8 : G7_StepPlus_V6;   // Step structure
      Trans8 : G7_TransitionPlus_V6;   // Transition structure
      Step9 : G7_StepPlus_V6;   // Step structure
      Trans9 : G7_TransitionPlus_V6;   // Transition structure
      Step10 : G7_StepPlus_V6;   // Step structure
      Trans10 : G7_TransitionPlus_V6;   // Transition structure
      Step11 : G7_StepPlus_V6;   // Step structure
      Step12 : G7_StepPlus_V6;   // Step structure
      Trans11 : G7_TransitionPlus_V6;   // Transition structure
      Step13 : G7_StepPlus_V6;   // Step structure
      Trans12 : G7_TransitionPlus_V6;   // Transition structure
      Step14 : G7_StepPlus_V6;   // Step structure
      Trans13 : G7_TransitionPlus_V6;   // Transition structure
      Step15 : G7_StepPlus_V6;   // Step structure
      Trans14 : G7_TransitionPlus_V6;   // Transition structure
      Trans15 : G7_TransitionPlus_V6;   // Transition structure
   END_VAR
BEGIN
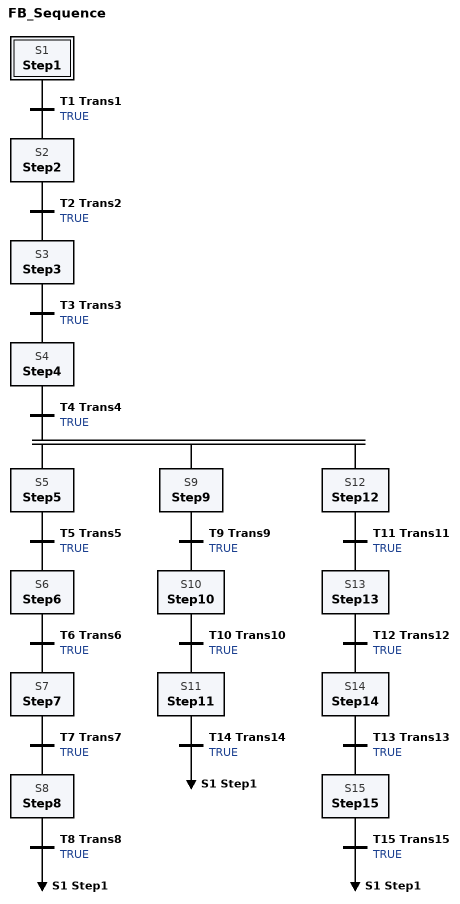
   // sequencer 1
   INITIAL_STEP Step1:   // S1, max time T#10S, warning time T#7S
   END_STEP
   TRANSITION Trans1 FROM Step1 TO Step2   // T1
      := TRUE;
   END_TRANSITION
   STEP Step2:   // S2, max time T#10S, warning time T#7S
   END_STEP
   TRANSITION Trans2 FROM Step2 TO Step3   // T2
      := TRUE;
   END_TRANSITION
   STEP Step3:   // S3, max time T#10S, warning time T#7S
   END_STEP
   TRANSITION Trans3 FROM Step3 TO Step4   // T3
      := TRUE;
   END_TRANSITION
   STEP Step4:   // S4, max time T#10S, warning time T#7S
   END_STEP
   TRANSITION Trans4 FROM Step4 TO (Step5, Step9, Step12)   // T4
      := TRUE;
   END_TRANSITION
   STEP Step5:   // S5, max time T#10S, warning time T#7S
   END_STEP
   TRANSITION Trans5 FROM Step5 TO Step6   // T5
      := TRUE;
   END_TRANSITION
   STEP Step6:   // S6, max time T#10S, warning time T#7S
   END_STEP
   TRANSITION Trans6 FROM Step6 TO Step7   // T6
      := TRUE;
   END_TRANSITION
   STEP Step7:   // S7, max time T#10S, warning time T#7S
   END_STEP
   TRANSITION Trans7 FROM Step7 TO Step8   // T7
      := TRUE;
   END_TRANSITION
   STEP Step8:   // S8, max time T#10S, warning time T#7S
   END_STEP
   TRANSITION Trans8 FROM Step8 TO Step1   // T8, jump
      := TRUE;
   END_TRANSITION
   STEP Step9:   // S9, max time T#10S, warning time T#7S
   END_STEP
   TRANSITION Trans9 FROM Step9 TO Step10   // T9
      := TRUE;
   END_TRANSITION
   STEP Step10:   // S10, max time T#10S, warning time T#7S
   END_STEP
   TRANSITION Trans10 FROM Step10 TO Step11   // T10
      := TRUE;
   END_TRANSITION
   STEP Step11:   // S11, max time T#10S, warning time T#7S
   END_STEP
   TRANSITION Trans14 FROM Step11 TO Step1   // T14, jump
      := TRUE;
   END_TRANSITION
   STEP Step12:   // S12, max time T#10S, warning time T#7S
   END_STEP
   TRANSITION Trans11 FROM Step12 TO Step13   // T11
      := TRUE;
   END_TRANSITION
   STEP Step13:   // S13, max time T#10S, warning time T#7S
   END_STEP
   TRANSITION Trans12 FROM Step13 TO Step14   // T12
      := TRUE;
   END_TRANSITION
   STEP Step14:   // S14, max time T#10S, warning time T#7S
   END_STEP
   TRANSITION Trans13 FROM Step14 TO Step15   // T13
      := TRUE;
   END_TRANSITION
   STEP Step15:   // S15, max time T#10S, warning time T#7S
   END_STEP
   TRANSITION Trans15 FROM Step15 TO Step1   // T15, jump
      := TRUE;
   END_TRANSITION
END_FUNCTION_BLOCK

FUNCTION "FC_Area" : Void   // FC1, LAD
{ S7_Optimized_Access := 'TRUE' }
VERSION : 0.1
BEGIN

REGION Network 1: Conveyor1
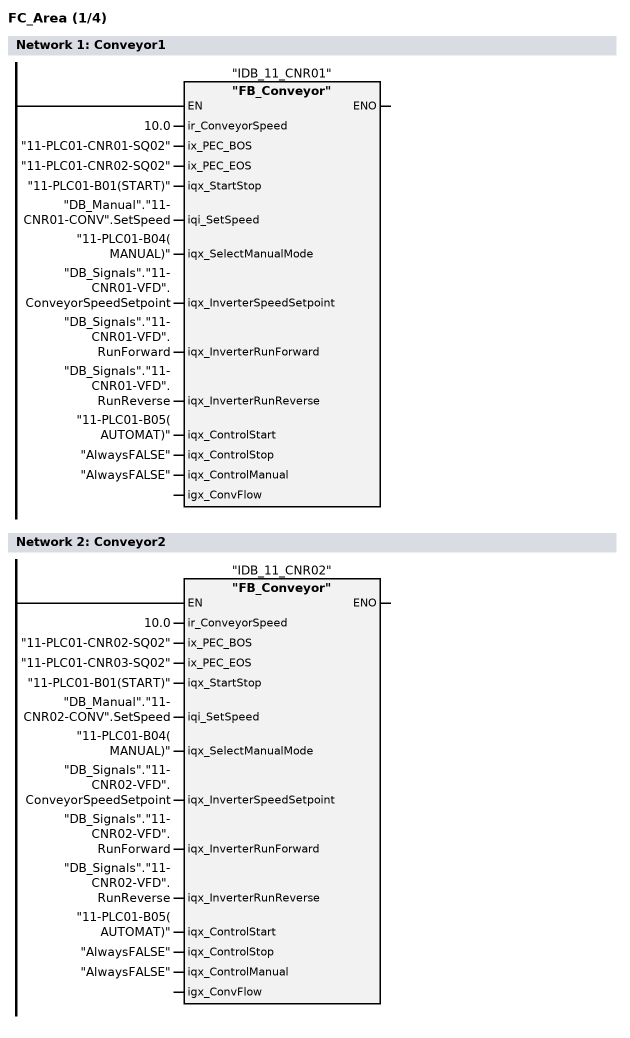
   RUNG wire#powerrail
      "IDB_11_CNR01"(ir_ConveyorSpeed := 10.0, ix_PEC_BOS := "11-PLC01-CNR01-SQ02", ix_PEC_EOS := "11-PLC01-CNR02-SQ02", iqx_StartStop := "11-PLC01-B01(START)", iqi_SetSpeed := "DB_Manual"."11-CNR01-CONV".SetSpeed, iqx_SelectManualMode := "11-PLC01-B04(MANUAL)", iqx_InverterSpeedSetpoint := "DB_Signals"."11-CNR01-VFD".ConveyorSpeedSetpoint, iqx_InverterRunForward := "DB_Signals"."11-CNR01-VFD".RunForward, iqx_InverterRunReverse := "DB_Signals"."11-CNR01-VFD".RunReverse, iqx_ControlStart := "11-PLC01-B05(AUTOMAT)", iqx_ControlStop := "AlwaysFALSE", iqx_ControlManual := "AlwaysFALSE", igx_ConvFlow :=)
   END_RUNG
   // the same network as SCL:
   "IDB_11_CNR01"(ir_ConveyorSpeed := 10.0,   // "FB_Conveyor"
                  ix_PEC_BOS := "11-PLC01-CNR01-SQ02",
                  ix_PEC_EOS := "11-PLC01-CNR02-SQ02",
                  iqx_StartStop := "11-PLC01-B01(START)",
                  iqi_SetSpeed := "DB_Manual"."11-CNR01-CONV".SetSpeed,
                  iqx_SelectManualMode := "11-PLC01-B04(MANUAL)",
                  iqx_InverterSpeedSetpoint := "DB_Signals"."11-CNR01-VFD".ConveyorSpeedSetpoint,
                  iqx_InverterRunForward := "DB_Signals"."11-CNR01-VFD".RunForward,
                  iqx_InverterRunReverse := "DB_Signals"."11-CNR01-VFD".RunReverse,
                  iqx_ControlStart := "11-PLC01-B05(AUTOMAT)",
                  iqx_ControlStop := "AlwaysFALSE",
                  iqx_ControlManual := "AlwaysFALSE");
END_REGION

REGION Network 2: Conveyor2
   RUNG wire#powerrail
      "IDB_11_CNR02"(ir_ConveyorSpeed := 10.0, ix_PEC_BOS := "11-PLC01-CNR02-SQ02", ix_PEC_EOS := "11-PLC01-CNR03-SQ02", iqx_StartStop := "11-PLC01-B01(START)", iqi_SetSpeed := "DB_Manual"."11-CNR02-CONV".SetSpeed, iqx_SelectManualMode := "11-PLC01-B04(MANUAL)", iqx_InverterSpeedSetpoint := "DB_Signals"."11-CNR02-VFD".ConveyorSpeedSetpoint, iqx_InverterRunForward := "DB_Signals"."11-CNR02-VFD".RunForward, iqx_InverterRunReverse := "DB_Signals"."11-CNR02-VFD".RunReverse, iqx_ControlStart := "11-PLC01-B05(AUTOMAT)", iqx_ControlStop := "AlwaysFALSE", iqx_ControlManual := "AlwaysFALSE", igx_ConvFlow :=)
   END_RUNG
   // the same network as SCL:
   "IDB_11_CNR02"(ir_ConveyorSpeed := 10.0,   // "FB_Conveyor"
                  ix_PEC_BOS := "11-PLC01-CNR02-SQ02",
                  ix_PEC_EOS := "11-PLC01-CNR03-SQ02",
                  iqx_StartStop := "11-PLC01-B01(START)",
                  iqi_SetSpeed := "DB_Manual"."11-CNR02-CONV".SetSpeed,
                  iqx_SelectManualMode := "11-PLC01-B04(MANUAL)",
                  iqx_InverterSpeedSetpoint := "DB_Signals"."11-CNR02-VFD".ConveyorSpeedSetpoint,
                  iqx_InverterRunForward := "DB_Signals"."11-CNR02-VFD".RunForward,
                  iqx_InverterRunReverse := "DB_Signals"."11-CNR02-VFD".RunReverse,
                  iqx_ControlStart := "11-PLC01-B05(AUTOMAT)",
                  iqx_ControlStop := "AlwaysFALSE",
                  iqx_ControlManual := "AlwaysFALSE");
END_REGION

REGION Network 3: Converyor3
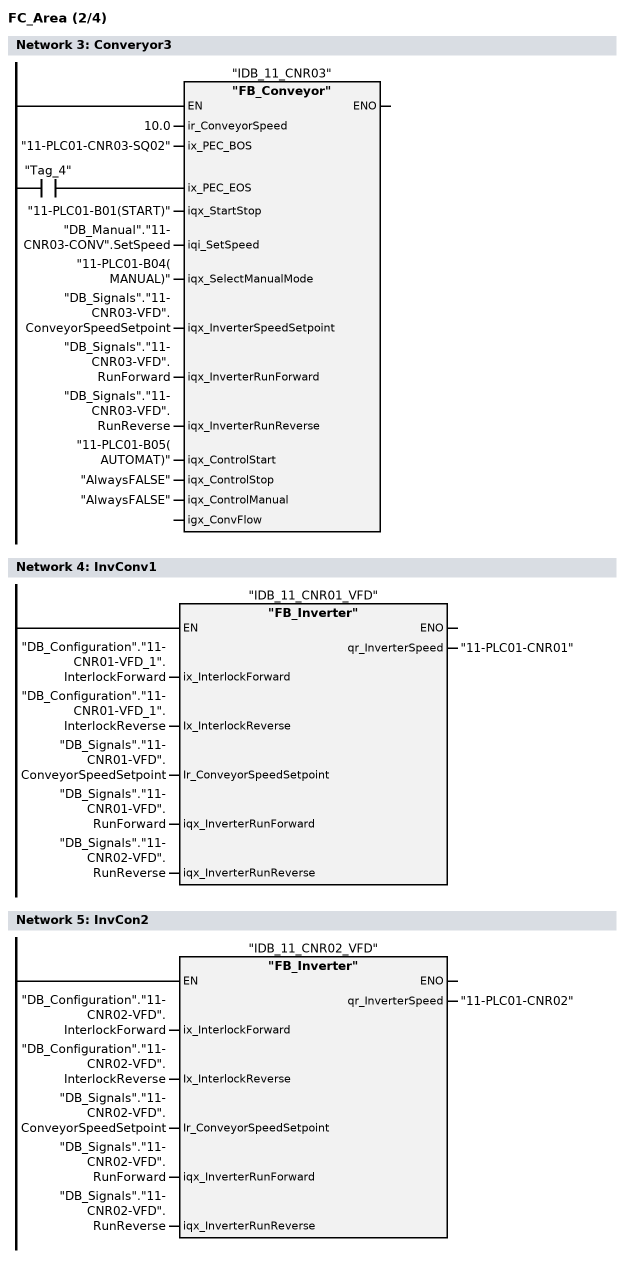
   RUNG wire#powerrail
      "IDB_11_CNR03"(ix_PEC_EOS := wire#w1, ir_ConveyorSpeed := 10.0, ix_PEC_BOS := "11-PLC01-CNR03-SQ02", iqx_StartStop := "11-PLC01-B01(START)", iqi_SetSpeed := "DB_Manual"."11-CNR03-CONV".SetSpeed, iqx_SelectManualMode := "11-PLC01-B04(MANUAL)", iqx_InverterSpeedSetpoint := "DB_Signals"."11-CNR03-VFD".ConveyorSpeedSetpoint, iqx_InverterRunForward := "DB_Signals"."11-CNR03-VFD".RunForward, iqx_InverterRunReverse := "DB_Signals"."11-CNR03-VFD".RunReverse, iqx_ControlStart := "11-PLC01-B05(AUTOMAT)", iqx_ControlStop := "AlwaysFALSE", iqx_ControlManual := "AlwaysFALSE", igx_ConvFlow :=)
   END_RUNG
   RUNG wire#powerrail
      Contact( "Tag_4" )
   END_RUNG wire#w1
   // the same network as SCL:
   "IDB_11_CNR03"(ir_ConveyorSpeed := 10.0,   // "FB_Conveyor"
                  ix_PEC_BOS := "11-PLC01-CNR03-SQ02",
                  ix_PEC_EOS := "Tag_4",
                  iqx_StartStop := "11-PLC01-B01(START)",
                  iqi_SetSpeed := "DB_Manual"."11-CNR03-CONV".SetSpeed,
                  iqx_SelectManualMode := "11-PLC01-B04(MANUAL)",
                  iqx_InverterSpeedSetpoint := "DB_Signals"."11-CNR03-VFD".ConveyorSpeedSetpoint,
                  iqx_InverterRunForward := "DB_Signals"."11-CNR03-VFD".RunForward,
                  iqx_InverterRunReverse := "DB_Signals"."11-CNR03-VFD".RunReverse,
                  iqx_ControlStart := "11-PLC01-B05(AUTOMAT)",
                  iqx_ControlStop := "AlwaysFALSE",
                  iqx_ControlManual := "AlwaysFALSE");
END_REGION

REGION Network 4: InvConv1
   RUNG wire#powerrail
      "IDB_11_CNR01_VFD"(ix_InterlockForward := "DB_Configuration"."11-CNR01-VFD_1".InterlockForward, Ix_InterlockReverse := "DB_Configuration"."11-CNR01-VFD_1".InterlockReverse, Ir_ConveyorSpeedSetpoint := "DB_Signals"."11-CNR01-VFD".ConveyorSpeedSetpoint, iqx_InverterRunForward := "DB_Signals"."11-CNR01-VFD".RunForward, iqx_InverterRunReverse := "DB_Signals"."11-CNR02-VFD".RunReverse, qr_InverterSpeed => "11-PLC01-CNR01")
   END_RUNG
   // the same network as SCL:
   "IDB_11_CNR01_VFD"(ix_InterlockForward := "DB_Configuration"."11-CNR01-VFD_1".InterlockForward,   // "FB_Inverter"
                      Ix_InterlockReverse := "DB_Configuration"."11-CNR01-VFD_1".InterlockReverse,
                      Ir_ConveyorSpeedSetpoint := "DB_Signals"."11-CNR01-VFD".ConveyorSpeedSetpoint,
                      iqx_InverterRunForward := "DB_Signals"."11-CNR01-VFD".RunForward,
                      iqx_InverterRunReverse := "DB_Signals"."11-CNR02-VFD".RunReverse,
                      qr_InverterSpeed => "11-PLC01-CNR01");
END_REGION

REGION Network 5: InvCon2
   RUNG wire#powerrail
      "IDB_11_CNR02_VFD"(ix_InterlockForward := "DB_Configuration"."11-CNR02-VFD".InterlockForward, Ix_InterlockReverse := "DB_Configuration"."11-CNR02-VFD".InterlockReverse, Ir_ConveyorSpeedSetpoint := "DB_Signals"."11-CNR02-VFD".ConveyorSpeedSetpoint, iqx_InverterRunForward := "DB_Signals"."11-CNR02-VFD".RunForward, iqx_InverterRunReverse := "DB_Signals"."11-CNR02-VFD".RunReverse, qr_InverterSpeed => "11-PLC01-CNR02")
   END_RUNG
   // the same network as SCL:
   "IDB_11_CNR02_VFD"(ix_InterlockForward := "DB_Configuration"."11-CNR02-VFD".InterlockForward,   // "FB_Inverter"
                      Ix_InterlockReverse := "DB_Configuration"."11-CNR02-VFD".InterlockReverse,
                      Ir_ConveyorSpeedSetpoint := "DB_Signals"."11-CNR02-VFD".ConveyorSpeedSetpoint,
                      iqx_InverterRunForward := "DB_Signals"."11-CNR02-VFD".RunForward,
                      iqx_InverterRunReverse := "DB_Signals"."11-CNR02-VFD".RunReverse,
                      qr_InverterSpeed => "11-PLC01-CNR02");
END_REGION

REGION Network 6: InvCon3
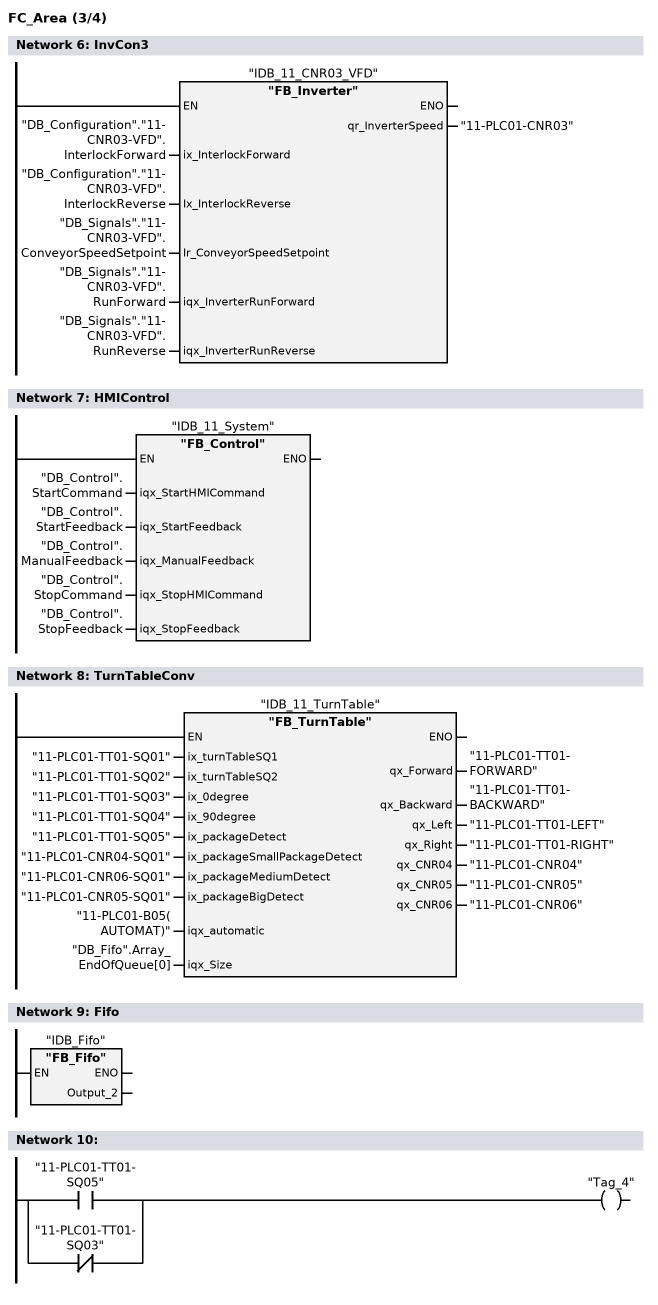
   RUNG wire#powerrail
      "IDB_11_CNR03_VFD"(ix_InterlockForward := "DB_Configuration"."11-CNR03-VFD".InterlockForward, Ix_InterlockReverse := "DB_Configuration"."11-CNR03-VFD".InterlockReverse, Ir_ConveyorSpeedSetpoint := "DB_Signals"."11-CNR03-VFD".ConveyorSpeedSetpoint, iqx_InverterRunForward := "DB_Signals"."11-CNR03-VFD".RunForward, iqx_InverterRunReverse := "DB_Signals"."11-CNR03-VFD".RunReverse, qr_InverterSpeed => "11-PLC01-CNR03")
   END_RUNG
   // the same network as SCL:
   "IDB_11_CNR03_VFD"(ix_InterlockForward := "DB_Configuration"."11-CNR03-VFD".InterlockForward,   // "FB_Inverter"
                      Ix_InterlockReverse := "DB_Configuration"."11-CNR03-VFD".InterlockReverse,
                      Ir_ConveyorSpeedSetpoint := "DB_Signals"."11-CNR03-VFD".ConveyorSpeedSetpoint,
                      iqx_InverterRunForward := "DB_Signals"."11-CNR03-VFD".RunForward,
                      iqx_InverterRunReverse := "DB_Signals"."11-CNR03-VFD".RunReverse,
                      qr_InverterSpeed => "11-PLC01-CNR03");
END_REGION

REGION Network 7: HMIControl
   RUNG wire#powerrail
      "IDB_11_System"(iqx_StartHMICommand := "DB_Control".StartCommand, iqx_StartFeedback := "DB_Control".StartFeedback, iqx_ManualFeedback := "DB_Control".ManualFeedback, iqx_StopHMICommand := "DB_Control".StopCommand, iqx_StopFeedback := "DB_Control".StopFeedback)
   END_RUNG
   // the same network as SCL:
   "IDB_11_System"(iqx_StartHMICommand := "DB_Control".StartCommand,   // "FB_Control"
                   iqx_StartFeedback := "DB_Control".StartFeedback,
                   iqx_ManualFeedback := "DB_Control".ManualFeedback,
                   iqx_StopHMICommand := "DB_Control".StopCommand,
                   iqx_StopFeedback := "DB_Control".StopFeedback);
END_REGION

REGION Network 8: TurnTableConv
   RUNG wire#powerrail
      "IDB_11_TurnTable"(ix_turnTableSQ1 := "11-PLC01-TT01-SQ01", ix_turnTableSQ2 := "11-PLC01-TT01-SQ02", ix_0degree := "11-PLC01-TT01-SQ03", ix_90degree := "11-PLC01-TT01-SQ04", ix_packageDetect := "11-PLC01-TT01-SQ05", ix_packageSmallPackageDetect := "11-PLC01-CNR04-SQ01", ix_packageMediumDetect := "11-PLC01-CNR06-SQ01", ix_packageBigDetect := "11-PLC01-CNR05-SQ01", iqx_automatic := "11-PLC01-B05(AUTOMAT)", iqx_Size := "DB_Fifo".Array_EndOfQueue[0], qx_Forward => "11-PLC01-TT01-FORWARD", qx_Backward => "11-PLC01-TT01-BACKWARD", qx_Left => "11-PLC01-TT01-LEFT", qx_Right => "11-PLC01-TT01-RIGHT", qx_CNR04 => "11-PLC01-CNR04", qx_CNR05 => "11-PLC01-CNR05", qx_CNR06 => "11-PLC01-CNR06")
   END_RUNG
   // the same network as SCL:
   "IDB_11_TurnTable"(ix_turnTableSQ1 := "11-PLC01-TT01-SQ01",   // "FB_TurnTable"
                      ix_turnTableSQ2 := "11-PLC01-TT01-SQ02",
                      ix_0degree := "11-PLC01-TT01-SQ03",
                      ix_90degree := "11-PLC01-TT01-SQ04",
                      ix_packageDetect := "11-PLC01-TT01-SQ05",
                      ix_packageSmallPackageDetect := "11-PLC01-CNR04-SQ01",
                      ix_packageMediumDetect := "11-PLC01-CNR06-SQ01",
                      ix_packageBigDetect := "11-PLC01-CNR05-SQ01",
                      iqx_automatic := "11-PLC01-B05(AUTOMAT)",
                      iqx_Size := "DB_Fifo".Array_EndOfQueue[0],
                      qx_Forward => "11-PLC01-TT01-FORWARD",
                      qx_Backward => "11-PLC01-TT01-BACKWARD",
                      qx_Left => "11-PLC01-TT01-LEFT",
                      qx_Right => "11-PLC01-TT01-RIGHT",
                      qx_CNR04 => "11-PLC01-CNR04",
                      qx_CNR05 => "11-PLC01-CNR05",
                      qx_CNR06 => "11-PLC01-CNR06");
END_REGION

REGION Network 9: Fifo
   RUNG wire#powerrail
      "IDB_Fifo"(Output_2 =>)
   END_RUNG
   // the same network as SCL:
   "IDB_Fifo"();   // "FB_Fifo"
END_REGION

REGION Network 10
   RUNG wire#powerrail
      Contact( "11-PLC01-TT01-SQ05" )
      wire#w1
      Coil( "Tag_4" )
   END_RUNG
   RUNG wire#powerrail
      I_Contact( "11-PLC01-TT01-SQ03" )
   END_RUNG wire#w1
   // the same network as SCL:
   "Tag_4" := "11-PLC01-TT01-SQ05" OR NOT "11-PLC01-TT01-SQ03";
END_REGION

REGION Network 11: Amount Of Package
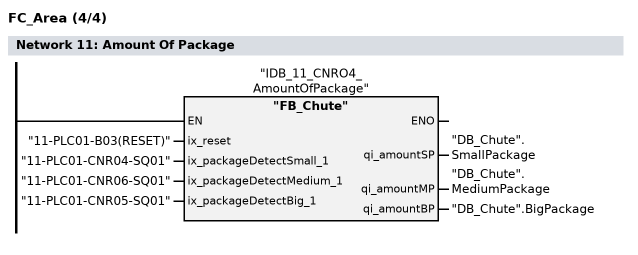
   RUNG wire#powerrail
      "IDB_11_CNRO4_AmountOfPackage"(ix_reset := "11-PLC01-B03(RESET)", ix_packageDetectSmall_1 := "11-PLC01-CNR04-SQ01", ix_packageDetectMedium_1 := "11-PLC01-CNR06-SQ01", ix_packageDetectBig_1 := "11-PLC01-CNR05-SQ01", qi_amountSP => "DB_Chute".SmallPackage, qi_amountMP => "DB_Chute".MediumPackage, qi_amountBP => "DB_Chute".BigPackage)
   END_RUNG
   // the same network as SCL:
   "IDB_11_CNRO4_AmountOfPackage"(ix_reset := "11-PLC01-B03(RESET)",   // "FB_Chute"
                           ix_packageDetectSmall_1 := "11-PLC01-CNR04-SQ01",
                           ix_packageDetectMedium_1 := "11-PLC01-CNR06-SQ01",
                           ix_packageDetectBig_1 := "11-PLC01-CNR05-SQ01",
                           qi_amountSP => "DB_Chute".SmallPackage,
                           qi_amountMP => "DB_Chute".MediumPackage,
                           qi_amountBP => "DB_Chute".BigPackage);
END_REGION
END_FUNCTION

ORGANIZATION_BLOCK "Main"   // OB1, LAD, ProgramCycle
TITLE = "Main Program Sweep (Cycle)"
{ S7_Optimized_Access := 'TRUE' }
VERSION : 0.1
   VAR_INPUT
      Initial_Call : Bool;   // Initial call of this OB
      Remanence : Bool;   // =True, if remanent data are available
   END_VAR
BEGIN

REGION Network 1
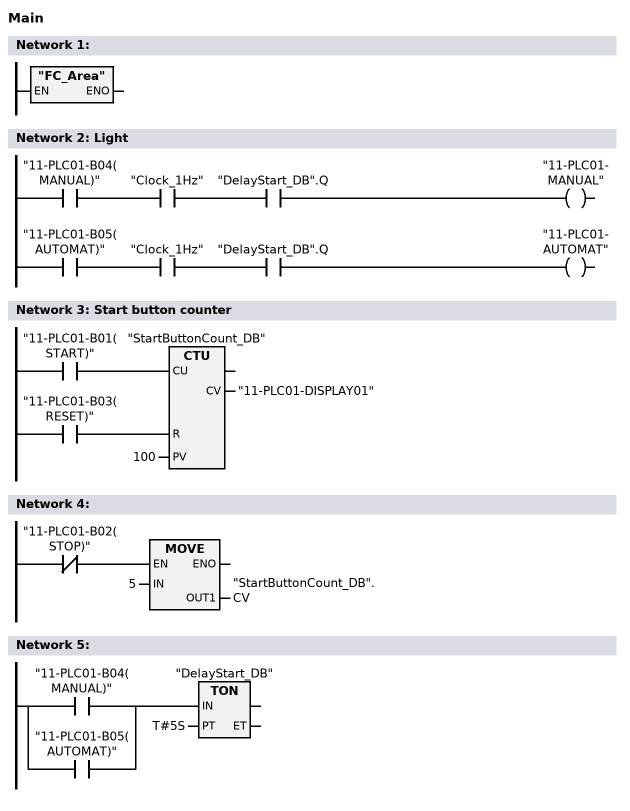
   RUNG wire#powerrail
      "FC_Area"()
   END_RUNG
   // the same network as SCL:
   "FC_Area"();
END_REGION

REGION Network 2: Light
   RUNG wire#powerrail
      Contact( "11-PLC01-B04(MANUAL)" )
      Contact( "Clock_1Hz" )
      Contact( "DelayStart_DB".Q )
      Coil( "11-PLC01-MANUAL" )
   END_RUNG
   RUNG wire#powerrail
      Contact( "11-PLC01-B05(AUTOMAT)" )
      Contact( "Clock_1Hz" )
      Contact( "DelayStart_DB".Q )
      Coil( "11-PLC01-AUTOMAT" )
   END_RUNG
   // the same network as SCL:
   "11-PLC01-MANUAL" := "11-PLC01-B04(MANUAL)" AND "Clock_1Hz" AND "DelayStart_DB".Q;
   "11-PLC01-AUTOMAT" := "11-PLC01-B05(AUTOMAT)" AND "Clock_1Hz" AND "DelayStart_DB".Q;
END_REGION

REGION Network 3: Start button counter
   "StartButtonCount_DB".CTU(CU := "11-PLC01-B01(START)",
                           R := "11-PLC01-B03(RESET)",
                           PV := 100,
                           CV => "11-PLC01-DISPLAY01");
END_REGION

REGION Network 4
   RUNG wire#powerrail
      I_Contact( "11-PLC01-B02(STOP)" )
      Move(in := 5, out1 => "StartButtonCount_DB".CV)
   END_RUNG
   // the same network as SCL:
   IF NOT "11-PLC01-B02(STOP)" THEN "StartButtonCount_DB".CV := 5; END_IF;
END_REGION

REGION Network 5
   "DelayStart_DB".TON(IN := "11-PLC01-B04(MANUAL)" OR "11-PLC01-B05(AUTOMAT)", PT := T#5S);
END_REGION
END_ORGANIZATION_BLOCK